LIN {X 0,Y 148.489,Z 220.439,A -85,B 0,C 180,E1 -25225.922,E2 -25225.922} C_VEL
LIN {X 0,Y 152.056,Z 225.38,A -85,B 0,C 180,E1 -25229.033,E2 -25229.033} C_VEL
LIN {X 0,Y 155.13,Z 229.793,A -85,B 0,C 180,E1 -25231.399,E2 -25231.399} C_VEL
LIN {X 0,Y 159.463,Z 236.417,A -85,B 0,C 180,E1 -25234.38,E2 -25234.38} C_VEL
LIN {X 0,Y 163.977,Z 245.373,A -85,B 0,C 180,E1 -25237.257,E2 -25237.257} C_VEL
LIN {X 0,Y 168.416,Z 255.821,A -85,B 0,C 180,E1 -25239.882,E2 -25239.882} C_VEL
LIN {X 0,Y 170.789,Z 262.4,A -85,B 0,C 180,E1 -25241.237,E2 -25241.237} C_VEL
LIN {X 0,Y 168.029,Z 299.799,A -85,B 0,C 180,E1 -25242.631,E2 -25242.631} C_VEL
LIN {X 0,Y 166.027,Z 312.888,A -85,B 0,C 180,E1 -25243.453,E2 -25243.453} C_VEL
LIN {X 0,Y 163.042,Z 325.855,A -85,B 0,C 180,E1 -25244.664,E2 -25244.664} C_VEL
LIN {X 0,Y 159.734,Z 336.912,A -85,B 0,C 180,E1 -25246.134,E2 -25246.134} C_VEL
LIN {X 0,Y 155.587,Z 348.447,A -85,B 0,C 180,E1 -25248.22,E2 -25248.22} C_VEL
LIN {X 0,Y 151.08,Z 358.834,A -85,B 0,C 180,E1 -25250.668,E2 -25250.668} C_VEL
LIN {X 0,Y 146.904,Z 367.324,A -85,B 0,C 180,E1 -25253.272,E2 -25253.272} C_VEL
LIN {X 0,Y 142.719,Z 375.157,A -85,B 0,C 180,E1 -25256.358,E2 -25256.358} C_VEL
LIN {X 0,Y 138.407,Z 382.806,A -85,B 0,C 180,E1 -25260.324,E2 -25260.324} C_VEL
LIN {X 0,Y 135.143,Z 388.047,A -85,B 0,C 180,E1 -25263.765,E2 -25263.765} C_VEL
LIN {X 0,Y 131.795,Z 393.123,A -85,B 0,C 180,E1 -25268.081,E2 -25268.081} C_VEL
LIN {X 0,Y 129.336,Z 397.065,A -85,B 0,C 180,E1 -25272.61,E2 -25272.61} C_VEL
LIN {X 0,Y 127.624,Z 399.977,A -85,B 0,C 180,E1 -25277.274,E2 -25277.274} C_VEL
LIN {X 0,Y 126.711,Z 401.714,A -85,B 0,C 180,E1 -25281.57,E2 -25281.57} C_VEL
LIN {X 0,Y 126.307,Z 402.951,A -85,B 0,C 180,E1 -25286.809,E2 -25286.809} C_VEL
LIN {X 0,Y 126.321,Z 403.159,A -85,B 0,C 180,E1 -25289.999,E2 -25289.999} C_VEL
LIN {X 0,Y 126.384,Z 402.517,A -85,B 0,C 180,E1 -25295.368,E2 -25295.368} C_VEL
LIN {X 0,Y 126.011,Z 401.88,A -85,B 0,C 180,E1 -25298.026,E2 -25298.026} C_VEL
LIN {X 0,Y 124.021,Z 400.249,A -85,B 0,C 180,E1 -25302.416,E2 -25302.416} C_VEL
LIN {X 0,Y 122.691,Z 398.422,A -85,B 0,C 180,E1 -25305.973,E2 -25305.973} C_VEL
LIN {X 0,Y 122.726,Z 396.742,A -85,B 0,C 180,E1 -25308.632,E2 -25308.632} C_VEL
LIN {X 0,Y 123.046,Z 396.081,A -85,B 0,C 180,E1 -25309.494,E2 -25309.494} C_VEL
LIN {X 0,Y 126.316,Z 391.361,A -85,B 0,C 180,E1 -25314.661,E2 -25314.661} C_VEL
LIN {X 0,Y 130.041,Z 385.839,A -85,B 0,C 180,E1 -25319.102,E2 -25319.102} C_VEL
LIN {X 0,Y 134.152,Z 379.389,A -85,B 0,C 180,E1 -25323.048,E2 -25323.048} C_VEL
LIN {X 0,Y 138.51,Z 371.906,A -85,B 0,C 180,E1 -25326.595,E2 -25326.595} C_VEL
LIN {X 0,Y 143.179,Z 363.415,A -85,B 0,C 180,E1 -25329.648,E2 -25329.648} C_VEL
LIN {X 0,Y 148.185,Z 352.923,A -85,B 0,C 180,E1 -25332.516,E2 -25332.516} C_VEL
LIN {X 0,Y 152.513,Z 342.536,A -85,B 0,C 180,E1 -25334.644,E2 -25334.644} C_VEL
LIN {X 0,Y 156.431,Z 331.134,A -85,B 0,C 180,E1 -25336.42,E2 -25336.42} C_VEL
LIN {X 0,Y 159.575,Z 319.369,A -85,B 0,C 180,E1 -25337.767,E2 -25337.767} C_VEL
LIN {X 0,Y 162.297,Z 305.659,A -85,B 0,C 180,E1 -25338.812,E2 -25338.812} C_VEL
LIN {X 0,Y 163.803,Z 292.635,A -85,B 0,C 180,E1 -25339.441,E2 -25339.441} C_VEL
LIN {X 0,Y 165.84,Z 264.469,A -85,B 0,C 180,E1 -25340.466,E2 -25340.466} C_VEL
LIN {X 0,Y 162.183,Z 254.665,A -85,B 0,C 180,E1 -25342.749,E2 -25342.749} C_VEL
LIN {X 0,Y 157.734,Z 244.687,A -85,B 0,C 180,E1 -25345.703,E2 -25345.703} C_VEL
LIN {X 0,Y 155.11,Z 239.926,A -85,B 0,C 180,E1 -25347.545,E2 -25347.545} C_VEL
LIN {X 0,Y 150.936,Z 233.432,A -85,B 0,C 180,E1 -25350.731,E2 -25350.731} C_VEL
LIN {X 0,Y 148.33,Z 229.665,A -85,B 0,C 180,E1 -25352.963,E2 -25352.963} C_VEL
LIN {X 0,Y 145.763,Z 225.988,A -85,B 0,C 180,E1 -25355.427,E2 -25355.427} C_VEL
LIN {X 0,Y 142.909,Z 222.259,A -85,B 0,C 180,E1 -25358.546,E2 -25358.546} C_VEL
LIN {X 0,Y 142.242,Z 221.258,A -85,B 0,C 180,E1 -25359.376,E2 -25359.376} C_VEL
LIN {X 0,Y 139.642,Z 218.363,A -85,B 0,C 180,E1 -25362.898,E2 -25362.898} C_VEL
LIN {X 0,Y 138.606,Z 216.213,A -85,B 0,C 180,E1 -25364.75,E2 -25364.75} C_VEL
LIN {X 0,Y 136.107,Z 214.124,A -85,B 0,C 180,E1 -25369.815,E2 -25369.815} C_VEL
LIN {X 0,Y 134.66,Z 211.097,A -85,B 0,C 180,E1 -25375.885,E2 -25375.885} C_VEL
LIN {X 0,Y 134.387,Z 210.372,A -85,B 0,C 180,E1 -25380,E2 -25380} C_VEL
LIN {X 0,Y 134.78,Z 211.442,A -85,B 0,C 180,E1 -25385.142,E2 -25385.142} C_VEL
LIN {X 0,Y 137.586,Z 215.64,A -85,B 0,C 180,E1 -25393.665,E2 -25393.665} C_VEL
LIN {X 0,Y 138.782,Z 216.531,A -85,B 0,C 180,E1 -25395.747,E2 -25395.747} C_VEL
LIN {X 0,Y 140.767,Z 219.894,A -85,B 0,C 180,E1 -25398.937,E2 -25398.937} C_VEL
LIN {X 0,Y 142.714,Z 221.837,A -85,B 0,C 180,E1 -25401.372,E2 -25401.372} C_VEL
LIN {X 0,Y 145.287,Z 225.513,A -85,B 0,C 180,E1 -25404.279,E2 -25404.279} C_VEL
LIN {X 0,Y 146.423,Z 226.871,A -85,B 0,C 180,E1 -25405.403,E2 -25405.403} C_VEL
LIN {X 0,Y 149.767,Z 231.675,A -85,B 0,C 180,E1 -25408.464,E2 -25408.464} C_VEL
LIN {X 0,Y 152.784,Z 236.265,A -85,B 0,C 180,E1 -25410.908,E2 -25410.908} C_VEL
LIN {X 0,Y 156.375,Z 241.912,A -85,B 0,C 180,E1 -25413.51,E2 -25413.51} C_VEL
LIN {X 0,Y 161.078,Z 250.32,A -85,B 0,C 180,E1 -25416.588,E2 -25416.588} C_VEL
LIN {X 0,Y 164.621,Z 258.823,A -85,B 0,C 180,E1 -25418.808,E2 -25418.808} C_VEL
LIN {X 0,Y 165.991,Z 262.553,A -85,B 0,C 180,E1 -25419.643,E2 -25419.643} C_VEL
LIN {X 0,Y 163.242,Z 297.955,A -85,B 0,C 180,E1 -25420.978,E2 -25420.978} C_VEL
LIN {X 0,Y 161.003,Z 311.512,A -85,B 0,C 180,E1 -25421.82,E2 -25421.82} C_VEL
LIN {X 0,Y 158.165,Z 324.036,A -85,B 0,C 180,E1 -25423.084,E2 -25423.084} C_VEL
LIN {X 0,Y 154.484,Z 335.831,A -85,B 0,C 180,E1 -25424.7,E2 -25424.7} C_VEL
LIN {X 0,Y 150.193,Z 347.172,A -85,B 0,C 180,E1 -25426.818,E2 -25426.818} C_VEL
LIN {X 0,Y 145.558,Z 357.394,A -85,B 0,C 180,E1 -25429.324,E2 -25429.324} C_VEL
LIN {X 0,Y 140.81,Z 366.572,A -85,B 0,C 180,E1 -25432.311,E2 -25432.311} C_VEL
LIN {X 0,Y 135.827,Z 375.493,A -85,B 0,C 180,E1 -25436.207,E2 -25436.207} C_VEL
LIN {X 0,Y 131.307,Z 382.676,A -85,B 0,C 180,E1 -25440.326,E2 -25440.326} C_VEL
LIN {X 0,Y 127.933,Z 387.52,A -85,B 0,C 180,E1 -25443.931,E2 -25443.931} C_VEL
LIN {X 0,Y 124.651,Z 392.227,A -85,B 0,C 180,E1 -25448.503,E2 -25448.503} C_VEL
LIN {X 0,Y 122.223,Z 395.828,A -85,B 0,C 180,E1 -25453.293,E2 -25453.293} C_VEL
LIN {X 0,Y 120.997,Z 397.687,A -85,B 0,C 180,E1 -25456.567,E2 -25456.567} C_VEL
LIN {X 0,Y 120.126,Z 399.083,A -85,B 0,C 180,E1 -25459.893,E2 -25459.893} C_VEL
LIN {X 0,Y 119.293,Z 400.686,A -85,B 0,C 180,E1 -25466.624,E2 -25466.624} C_VEL
LIN {X 0,Y 119.281,Z 400.912,A -85,B 0,C 180,E1 -25470.001,E2 -25470.001} C_VEL
LIN {X 0,Y 119.293,Z 400.715,A -85,B 0,C 180,E1 -25473.379,E2 -25473.379} C_VEL
LIN {X 0,Y 120.127,Z 399.15,A -85,B 0,C 180,E1 -25480.11,E2 -25480.11} C_VEL
LIN {X 0,Y 120.997,Z 397.783,A -85,B 0,C 180,E1 -25483.436,E2 -25483.436} C_VEL
LIN {X 0,Y 122.934,Z 394.897,A -85,B 0,C 180,E1 -25488.327,E2 -25488.327} C_VEL
LIN {X 0,Y 125.547,Z 390.986,A -85,B 0,C 180,E1 -25493.071,E2 -25493.071} C_VEL
LIN {X 0,Y 129.152,Z 385.94,A -85,B 0,C 180,E1 -25497.552,E2 -25497.552} C_VEL
LIN {X 0,Y 133.341,Z 379.586,A -85,B 0,C 180,E1 -25501.808,E2 -25501.808} C_VEL
LIN {X 0,Y 138.101,Z 371.645,A -85,B 0,C 180,E1 -25505.819,E2 -25505.819} C_VEL
LIN {X 0,Y 142.511,Z 363.544,A -85,B 0,C 180,E1 -25508.96,E2 -25508.96} C_VEL
LIN {X 0,Y 147.519,Z 353.661,A -85,B 0,C 180,E1 -25511.835,E2 -25511.835} C_VEL
LIN {X 0,Y 152.249,Z 342.531,A -85,B 0,C 180,E1 -25514.282,E2 -25514.282} C_VEL
LIN {X 0,Y 156.034,Z 331.622,A -85,B 0,C 180,E1 -25516.109,E2 -25516.109} C_VEL
LIN {X 0,Y 159.484,Z 319.56,A -85,B 0,C 180,E1 -25517.572,E2 -25517.572} C_VEL
LIN {X 0,Y 162.175,Z 306.48,A -85,B 0,C 180,E1 -25518.694,E2 -25518.694} C_VEL
LIN {X 0,Y 163.866,Z 293.691,A -85,B 0,C 180,E1 -25519.374,E2 -25519.374} C_VEL
LIN {X 0,Y 166.138,Z 262.629,A -85,B 0,C 180,E1 -25520.526,E2 -25520.526} C_VEL
LIN {X 0,Y 162.62,Z 253.552,A -85,B 0,C 180,E1 -25522.703,E2 -25522.703} C_VEL
LIN {X 0,Y 159.851,Z 247.737,A -85,B 0,C 180,E1 -25524.466,E2 -25524.466} C_VEL
LIN {X 0,Y 154.056,Z 237.994,A -85,B 0,C 180,E1 -25528.452,E2 -25528.452} C_VEL
LIN {X 0,Y 149.123,Z 230.481,A -85,B 0,C 180,E1 -25532.454,E2 -25532.454} C_VEL
LIN {X 0,Y 145.784,Z 225.926,A -85,B 0,C 180,E1 -25535.62,E2 -25535.62} C_VEL
LIN {X 0,Y 143.1,Z 222.493,A -85,B 0,C 180,E1 -25538.575,E2 -25538.575} C_VEL
LIN {X 0,Y 142.318,Z 221.292,A -85,B 0,C 180,E1 -25539.564,E2 -25539.564} C_VEL
LIN {X 0,Y 139.639,Z 218.207,A -85,B 0,C 180,E1 -25543.296,E2 -25543.296} C_VEL
LIN {X 0,Y 138.742,Z 216.293,A -85,B 0,C 180,E1 -25544.953,E2 -25544.953} C_VEL
LIN {X 0,Y 135.941,Z 213.85,A -85,B 0,C 180,E1 -25551.077,E2 -25551.077} C_VEL
LIN {X 0,Y 134.761,Z 210.99,A -85,B 0,C 180,E1 -25557.758,E2 -25557.758} C_VEL
LIN {X 0,Y 134.713,Z 210.681,A -85,B 0,C 180,E1 -25560.747,E2 -25560.747} C_VEL
LIN {X 0,Y 134.979,Z 211.831,A -85,B 0,C 180,E1 -25564.479,E2 -25564.479} C_VEL
LIN {X 0,Y 137.967,Z 215.899,A -85,B 0,C 180,E1 -25573.627,E2 -25573.627} C_VEL
LIN {X 0,Y 138.803,Z 216.447,A -85,B 0,C 180,E1 -25575.087,E2 -25575.087} C_VEL
LIN {X 0,Y 140.718,Z 219.788,A -85,B 0,C 180,E1 -25578.283,E2 -25578.283} C_VEL
LIN {X 0,Y 142.808,Z 221.926,A -85,B 0,C 180,E1 -25580.962,E2 -25580.962} C_VEL
LIN {X 0,Y 145.247,Z 225.428,A -85,B 0,C 180,E1 -25583.764,E2 -25583.764} C_VEL
LIN {X 0,Y 146.569,Z 227.031,A -85,B 0,C 180,E1 -25585.091,E2 -25585.091} C_VEL
LIN {X 0,Y 149.847,Z 231.734,A -85,B 0,C 180,E1 -25588.114,E2 -25588.114} C_VEL
LIN {X 0,Y 153.25,Z 236.86,A -85,B 0,C 180,E1 -25590.868,E2 -25590.868} C_VEL
LIN {X 0,Y 157.046,Z 243.057,A -85,B 0,C 180,E1 -25593.612,E2 -25593.612} C_VEL
LIN {X 0,Y 161.42,Z 252.589,A -85,B 0,C 180,E1 -25596.579,E2 -25596.579} C_VEL
LIN {X 0,Y 165.179,Z 262.134,A -85,B 0,C 180,E1 -25598.95,E2 -25598.95} C_VEL
LIN {X 0,Y 166.024,Z 264.644,A -85,B 0,C 180,E1 -25599.476,E2 -25599.476} C_VEL
LIN {X 0,Y 163.281,Z 299.957,A -85,B 0,C 180,E1 -25600.81,E2 -25600.81} C_VEL
LIN {X 0,Y 161.16,Z 313.156,A -85,B 0,C 180,E1 -25601.644,E2 -25601.644} C_VEL
LIN {X 0,Y 158.144,Z 325.797,A -85,B 0,C 180,E1 -25602.839,E2 -25602.839} C_VEL
LIN {X 0,Y 154.699,Z 336.852,A -85,B 0,C 180,E1 -25604.314,E2 -25604.314} C_VEL
LIN {X 0,Y 150.368,Z 348.386,A -85,B 0,C 180,E1 -25606.418,E2 -25606.418} C_VEL
LIN {X 0,Y 145.665,Z 358.772,A -85,B 0,C 180,E1 -25608.9,E2 -25608.9} C_VEL
LIN {X 0,Y 141.276,Z 367.262,A -85,B 0,C 180,E1 -25611.55,E2 -25611.55} C_VEL
LIN {X 0,Y 136.015,Z 376.462,A -85,B 0,C 180,E1 -25615.362,E2 -25615.362} C_VEL
LIN {X 0,Y 131.525,Z 383.859,A -85,B 0,C 180,E1 -25619.493,E2 -25619.493} C_VEL
LIN {X 0,Y 127.531,Z 389.797,A -85,B 0,C 180,E1 -25623.84,E2 -25623.84} C_VEL
LIN {X 0,Y 124.214,Z 394.486,A -85,B 0,C 180,E1 -25628.421,E2 -25628.421} C_VEL
LIN {X 0,Y 121.847,Z 398.067,A -85,B 0,C 180,E1 -25633.237,E2 -25633.237} C_VEL
LIN {X 0,Y 120.689,Z 399.913,A -85,B 0,C 180,E1 -25636.529,E2 -25636.529} C_VEL
LIN {X 0,Y 119.43,Z 402.284,A -85,B 0,C 180,E1 -25643.24,E2 -25643.24} C_VEL
LIN {X 0,Y 119.225,Z 402.886,A -85,B 0,C 180,E1 -25646.619,E2 -25646.619} C_VEL
LIN {X 0,Y 119.234,Z 403.094,A -85,B 0,C 180,E1 -25649.999,E2 -25649.999} C_VEL
LIN {X 0,Y 119.303,Z 402.488,A -85,B 0,C 180,E1 -25655.484,E2 -25655.484} C_VEL
LIN {X 0,Y 119.887,Z 401.259,A -85,B 0,C 180,E1 -25660.127,E2 -25660.127} C_VEL
LIN {X 0,Y 120.704,Z 399.859,A -85,B 0,C 180,E1 -25663.466,E2 -25663.466} C_VEL
LIN {X 0,Y 123.046,Z 396.081,A -85,B 0,C 180,E1 -25669.494,E2 -25669.494} C_VEL
LIN {X 0,Y 123.774,Z 394.072,A -85,B 0,C 180,E1 -25672.05,E2 -25672.05} C_VEL
LIN {X 0,Y 123.81,Z 390.329,A -85,B 0,C 180,E1 -25676.3,E2 -25676.3} C_VEL
LIN {X 0,Y 124.391,Z 385.968,A -85,B 0,C 180,E1 -25680.398,E2 -25680.398} C_VEL
LIN {X 0,Y 125.914,Z 382.924,A -85,B 0,C 180,E1 -25682.618,E2 -25682.618} C_VEL
LIN {X 0,Y 131.063,Z 374.812,A -85,B 0,C 180,E1 -25687.101,E2 -25687.101} C_VEL
LIN {X 0,Y 135.761,Z 366.932,A -85,B 0,C 180,E1 -25690.32,E2 -25690.32} C_VEL
LIN {X 0,Y 140.867,Z 357.317,A -85,B 0,C 180,E1 -25693.311,E2 -25693.311} C_VEL
LIN {X 0,Y 145.774,Z 346.644,A -85,B 0,C 180,E1 -25695.816,E2 -25695.816} C_VEL
LIN {X 0,Y 149.829,Z 336.315,A -85,B 0,C 180,E1 -25697.625,E2 -25697.625} C_VEL
LIN {X 0,Y 153.705,Z 323.946,A -85,B 0,C 180,E1 -25699.224,E2 -25699.224} C_VEL
LIN {X 0,Y 156.725,Z 311.132,A -85,B 0,C 180,E1 -25700.38,E2 -25700.38} C_VEL
LIN {X 0,Y 158.79,Z 297.868,A -85,B 0,C 180,E1 -25701.159,E2 -25701.159} C_VEL
LIN {X 0,Y 161.234,Z 266.782,A -85,B 0,C 180,E1 -25702.322,E2 -25702.322} C_VEL
LIN {X 0,Y 157.654,Z 257.066,A -85,B 0,C 180,E1 -25704.778,E2 -25704.778} C_VEL
LIN {X 0,Y 153.773,Z 248.275,A -85,B 0,C 180,E1 -25707.616,E2 -25707.616} C_VEL
LIN {X 0,Y 150.126,Z 242.029,A -85,B 0,C 180,E1 -25710.46,E2 -25710.46} C_VEL
LIN {X 0,Y 146.642,Z 236.472,A -85,B 0,C 180,E1 -25713.541,E2 -25713.541} C_VEL
LIN {X 0,Y 143.63,Z 232.219,A -85,B 0,C 180,E1 -25716.574,E2 -25716.574} C_VEL
LIN {X 0,Y 140.558,Z 227.87,A -85,B 0,C 180,E1 -25720.275,E2 -25720.275} C_VEL
LIN {X 0,Y 137.868,Z 224.441,A -85,B 0,C 180,E1 -25724.287,E2 -25724.287} C_VEL
LIN {X 0,Y 137.228,Z 223.045,A -85,B 0,C 180,E1 -25725.542,E2 -25725.542} C_VEL
LIN {X 0,Y 134.693,Z 220.54,A -85,B 0,C 180,E1 -25731.373,E2 -25731.373} C_VEL
LIN {X 0,Y 133.719,Z 218.034,A -85,B 0,C 180,E1 -25736.422,E2 -25736.422} C_VEL
LIN {X 0,Y 133.52,Z 217.429,A -85,B 0,C 180,E1 -25740,E2 -25740} C_VEL
LIN {X 0,Y 133.863,Z 218.47,A -85,B 0,C 180,E1 -25744.894,E2 -25744.894} C_VEL
LIN {X 0,Y 136.363,Z 222.503,A -85,B 0,C 180,E1 -25753.031,E2 -25753.031} C_VEL
LIN {X 0,Y 137.429,Z 223.408,A -85,B 0,C 180,E1 -25755.023,E2 -25755.023} C_VEL
LIN {X 0,Y 139.535,Z 226.869,A -85,B 0,C 180,E1 -25758.539,E2 -25758.539} C_VEL
LIN {X 0,Y 141.056,Z 228.526,A -85,B 0,C 180,E1 -25760.547,E2 -25760.547} C_VEL
LIN {X 0,Y 143.805,Z 232.367,A -85,B 0,C 180,E1 -25763.778,E2 -25763.778} C_VEL
LIN {X 0,Y 147.492,Z 237.884,A -85,B 0,C 180,E1 -25767.434,E2 -25767.434} C_VEL
LIN {X 0,Y 150.332,Z 242.336,A -85,B 0,C 180,E1 -25769.88,E2 -25769.88} C_VEL
LIN {X 0,Y 155.024,Z 250.278,A -85,B 0,C 180,E1 -25773.443,E2 -25773.443} C_VEL
LIN {X 0,Y 158.233,Z 256.652,A -85,B 0,C 180,E1 -25775.659,E2 -25775.659} C_VEL
LIN {X 0,Y 161.38,Z 264.879,A -85,B 0,C 180,E1 -25777.784,E2 -25777.784} C_VEL
LIN {X 0,Y 158.734,Z 297.656,A -85,B 0,C 180,E1 -25779.026,E2 -25779.026} C_VEL
LIN {X 0,Y 156.442,Z 311.248,A -85,B 0,C 180,E1 -25779.862,E2 -25779.862} C_VEL
LIN {X 0,Y 153.411,Z 324.107,A -85,B 0,C 180,E1 -25781.15,E2 -25781.15} C_VEL
LIN {X 0,Y 149.581,Z 335.901,A -85,B 0,C 180,E1 -25782.769,E2 -25782.769} C_VEL
LIN {X 0,Y 145.106,Z 347.241,A -85,B 0,C 180,E1 -25784.903,E2 -25784.903} C_VEL
LIN {X 0,Y 140.253,Z 357.463,A -85,B 0,C 180,E1 -25787.434,E2 -25787.434} C_VEL
LIN {X 0,Y 135.256,Z 366.64,A -85,B 0,C 180,E1 -25790.47,E2 -25790.47} C_VEL
LIN {X 0,Y 130.16,Z 375.252,A -85,B 0,C 180,E1 -25794.304,E2 -25794.304} C_VEL
LIN {X 0,Y 125.175,Z 382.743,A -85,B 0,C 180,E1 -25798.714,E2 -25798.714} C_VEL
LIN {X 0,Y 121.578,Z 387.587,A -85,B 0,C 180,E1 -25802.457,E2 -25802.457} C_VEL
LIN {X 0,Y 118.039,Z 392.294,A -85,B 0,C 180,E1 -25807.234,E2 -25807.234} C_VEL
LIN {X 0,Y 115.428,Z 395.894,A -85,B 0,C 180,E1 -25812.278,E2 -25812.278} C_VEL
LIN {X 0,Y 114.081,Z 397.753,A -85,B 0,C 180,E1 -25815.736,E2 -25815.736} C_VEL
LIN {X 0,Y 113.129,Z 399.148,A -85,B 0,C 180,E1 -25819.261,E2 -25819.261} C_VEL
LIN {X 0,Y 112.213,Z 400.751,A -85,B 0,C 180,E1 -25826.411,E2 -25826.411} C_VEL
LIN {X 0,Y 112.2,Z 400.977,A -85,B 0,C 180,E1 -25830.002,E2 -25830.002} C_VEL
LIN {X 0,Y 112.213,Z 400.78,A -85,B 0,C 180,E1 -25833.592,E2 -25833.592} C_VEL
LIN {X 0,Y 113.129,Z 399.215,A -85,B 0,C 180,E1 -25840.742,E2 -25840.742} C_VEL
LIN {X 0,Y 114.081,Z 397.848,A -85,B 0,C 180,E1 -25844.267,E2 -25844.267} C_VEL
LIN {X 0,Y 116.19,Z 394.962,A -85,B 0,C 180,E1 -25849.433,E2 -25849.433} C_VEL
LIN {X 0,Y 119.034,Z 391.05,A -85,B 0,C 180,E1 -25854.413,E2 -25854.413} C_VEL
LIN {X 0,Y 122.896,Z 386.003,A -85,B 0,C 180,E1 -25859.084,E2 -25859.084} C_VEL
LIN {X 0,Y 127.368,Z 379.649,A -85,B 0,C 180,E1 -25863.49,E2 -25863.49} C_VEL
LIN {X 0,Y 132.384,Z 371.704,A -85,B 0,C 180,E1 -25867.627,E2 -25867.627} C_VEL
LIN {X 0,Y 137.066,Z 363.606,A -85,B 0,C 180,E1 -25870.826,E2 -25870.826} C_VEL
LIN {X 0,Y 142.291,Z 353.723,A -85,B 0,C 180,E1 -25873.748,E2 -25873.748} C_VEL
LIN {X 0,Y 147.252,Z 342.591,A -85,B 0,C 180,E1 -25876.21,E2 -25876.21} C_VEL
LIN {X 0,Y 151.206,Z 331.682,A -85,B 0,C 180,E1 -25878.046,E2 -25878.046} C_VEL
LIN {X 0,Y 154.775,Z 319.618,A -85,B 0,C 180,E1 -25879.516,E2 -25879.516} C_VEL
LIN {X 0,Y 157.562,Z 306.663,A -85,B 0,C 180,E1 -25880.623,E2 -25880.623} C_VEL
LIN {X 0,Y 159.349,Z 293.381,A -85,B 0,C 180,E1 -25881.335,E2 -25881.335} C_VEL
LIN {X 0,Y 161.54,Z 264.943,A -85,B 0,C 180,E1 -25882.388,E2 -25882.388} C_VEL
LIN {X 0,Y 157.819,Z 255.359,A -85,B 0,C 180,E1 -25884.918,E2 -25884.918} C_VEL
LIN {X 0,Y 153.237,Z 246.935,A -85,B 0,C 180,E1 -25888.168,E2 -25888.168} C_VEL
LIN {X 0,Y 148.476,Z 239.258,A -85,B 0,C 180,E1 -25892.036,E2 -25892.036} C_VEL
LIN {X 0,Y 146.101,Z 235.699,A -85,B 0,C 180,E1 -25894.24,E2 -25894.24} C_VEL
LIN {X 0,Y 143.821,Z 232.339,A -85,B 0,C 180,E1 -25896.607,E2 -25896.607} C_VEL
LIN {X 0,Y 141.03,Z 228.357,A -85,B 0,C 180,E1 -25899.964,E2 -25899.964} C_VEL
LIN {X 0,Y 138.048,Z 224.594,A -85,B 0,C 180,E1 -25904.403,E2 -25904.403} C_VEL
LIN {X 0,Y 137.378,Z 223.109,A -85,B 0,C 180,E1 -25905.747,E2 -25905.747} C_VEL
LIN {X 0,Y 134.751,Z 220.492,A -85,B 0,C 180,E1 -25912.131,E2 -25912.131} C_VEL
LIN {X 0,Y 133.891,Z 218.08,A -85,B 0,C 180,E1 -25917.744,E2 -25917.744} C_VEL
LIN {X 0,Y 133.845,Z 217.746,A -85,B 0,C 180,E1 -25920.752,E2 -25920.752} C_VEL
LIN {X 0,Y 134.151,Z 219.184,A -85,B 0,C 180,E1 -25924.883,E2 -25924.883} C_VEL
LIN {X 0,Y 136.929,Z 222.866,A -85,B 0,C 180,E1 -25933.354,E2 -25933.354} C_VEL
LIN {X 0,Y 137.544,Z 223.498,A -85,B 0,C 180,E1 -25934.518,E2 -25934.518} C_VEL
LIN {X 0,Y 139.554,Z 226.828,A -85,B 0,C 180,E1 -25937.966,E2 -25937.966} C_VEL
LIN {X 0,Y 141.146,Z 228.577,A -85,B 0,C 180,E1 -25940.113,E2 -25940.113} C_VEL
LIN {X 0,Y 143.734,Z 232.244,A -85,B 0,C 180,E1 -25943.217,E2 -25943.217} C_VEL
LIN {X 0,Y 147.59,Z 237.946,A -85,B 0,C 180,E1 -25947.087,E2 -25947.087} C_VEL
LIN {X 0,Y 151.393,Z 243.842,A -85,B 0,C 180,E1 -25950.321,E2 -25950.321} C_VEL
LIN {X 0,Y 154.182,Z 248.936,A -85,B 0,C 180,E1 -25952.481,E2 -25952.481} C_VEL
LIN {X 0,Y 157.857,Z 257.311,A -85,B 0,C 180,E1 -25955.169,E2 -25955.169} C_VEL
LIN {X 0,Y 161.263,Z 266.348,A -85,B 0,C 180,E1 -25957.501,E2 -25957.501} C_VEL
LIN {X 0,Y 161.479,Z 267.017,A -85,B 0,C 180,E1 -25957.648,E2 -25957.648} C_VEL
LIN {X 0,Y 158.755,Z 299.84,A -85,B 0,C 180,E1 -25958.873,E2 -25958.873} C_VEL
LIN {X 0,Y 156.464,Z 313.428,A -85,B 0,C 180,E1 -25959.726,E2 -25959.726} C_VEL
LIN {X 0,Y 153.413,Z 325.738,A -85,B 0,C 180,E1 -25960.897,E2 -25960.897} C_VEL
LIN {X 0,Y 149.228,Z 338.374,A -85,B 0,C 180,E1 -25962.619,E2 -25962.619} C_VEL
LIN {X 0,Y 144.763,Z 349.618,A -85,B 0,C 180,E1 -25964.763,E2 -25964.763} C_VEL
LIN {X 0,Y 139.86,Z 359.74,A -85,B 0,C 180,E1 -25967.282,E2 -25967.282} C_VEL
LIN {X 0,Y 134.81,Z 368.862,A -85,B 0,C 180,E1 -25970.31,E2 -25970.31} C_VEL
LIN {X 0,Y 129.465,Z 377.601,A -85,B 0,C 180,E1 -25974.189,E2 -25974.189} C_VEL
LIN {X 0,Y 124.666,Z 384.906,A -85,B 0,C 180,E1 -25978.569,E2 -25978.569} C_VEL
LIN {X 0,Y 119.893,Z 391.415,A -85,B 0,C 180,E1 -25983.918,E2 -25983.918} C_VEL
LIN {X 0,Y 116.622,Z 395.721,A -85,B 0,C 180,E1 -25988.802,E2 -25988.802} C_VEL
LIN {X 0,Y 115.053,Z 398.003,A -85,B 0,C 180,E1 -25992.215,E2 -25992.215} C_VEL
LIN {X 0,Y 113.772,Z 399.848,A -85,B 0,C 180,E1 -25995.693,E2 -25995.693} C_VEL
LIN {X 0,Y 112.36,Z 402.22,A -85,B 0,C 180,E1 -26002.812,E2 -26002.812} C_VEL
LIN {X 0,Y 112.135,Z 402.822,A -85,B 0,C 180,E1 -26006.405,E2 -26006.405} C_VEL
LIN {X 0,Y 112.139,Z 403.03,A -85,B 0,C 180,E1 -26009.998,E2 -26009.998} C_VEL
LIN {X 0,Y 112.135,Z 402.805,A -85,B 0,C 180,E1 -26013.592,E2 -26013.592} C_VEL
LIN {X 0,Y 112.359,Z 402.192,A -85,B 0,C 180,E1 -26017.185,E2 -26017.185} C_VEL
LIN {X 0,Y 112.895,Z 401.193,A -85,B 0,C 180,E1 -26020.762,E2 -26020.762} C_VEL
LIN {X 0,Y 113.784,Z 399.793,A -85,B 0,C 180,E1 -26024.302,E2 -26024.302} C_VEL
LIN {X 0,Y 116.164,Z 396.283,A -85,B 0,C 180,E1 -26030.296,E2 -26030.296} C_VEL
LIN {X 0,Y 119.885,Z 391.294,A -85,B 0,C 180,E1 -26036.08,E2 -26036.08} C_VEL
LIN {X 0,Y 123.881,Z 385.773,A -85,B 0,C 180,E1 -26040.7,E2 -26040.7} C_VEL
LIN {X 0,Y 125.914,Z 382.924,A -85,B 0,C 180,E1 -26042.618,E2 -26042.618} C_VEL
LIN {X 0,Y 127.508,Z 379.706,A -85,B 0,C 180,E1 -26044.738,E2 -26044.738} C_VEL
LIN {X 0,Y 128.744,Z 374.105,A -85,B 0,C 180,E1 -26048.355,E2 -26048.355} C_VEL
LIN {X 0,Y 130.262,Z 368.002,A -85,B 0,C 180,E1 -26051.719,E2 -26051.719} C_VEL
LIN {X 0,Y 132.2,Z 363.87,A -85,B 0,C 180,E1 -26053.37,E2 -26053.37} C_VEL
LIN {X 0,Y 137.478,Z 353.96,A -85,B 0,C 180,E1 -26056.224,E2 -26056.224} C_VEL
LIN {X 0,Y 142.164,Z 343.824,A -85,B 0,C 180,E1 -26058.39,E2 -26058.39} C_VEL
LIN {X 0,Y 146.387,Z 332.763,A -85,B 0,C 180,E1 -26060.185,E2 -26060.185} C_VEL
LIN {X 0,Y 150.098,Z 320.479,A -85,B 0,C 180,E1 -26061.651,E2 -26061.651} C_VEL
LIN {X 0,Y 153.106,Z 306.849,A -85,B 0,C 180,E1 -26062.715,E2 -26062.715} C_VEL
LIN {X 0,Y 154.809,Z 293.931,A -85,B 0,C 180,E1 -26063.375,E2 -26063.375} C_VEL
LIN {X 0,Y 156.789,Z 269.085,A -85,B 0,C 180,E1 -26064.294,E2 -26064.294} C_VEL
LIN {X 0,Y 153.223,Z 259.353,A -85,B 0,C 180,E1 -26066.997,E2 -26066.997} C_VEL
LIN {X 0,Y 150.007,Z 252.084,A -85,B 0,C 180,E1 -26069.598,E2 -26069.598} C_VEL
LIN {X 0,Y 145.981,Z 245.196,A -85,B 0,C 180,E1 -26073.122,E2 -26073.122} C_VEL
LIN {X 0,Y 142.959,Z 240.534,A -85,B 0,C 180,E1 -26076.169,E2 -26076.169} C_VEL
LIN {X 0,Y 141.47,Z 238.323,A -85,B 0,C 180,E1 -26077.857,E2 -26077.857} C_VEL
LIN {X 0,Y 138.858,Z 234.383,A -85,B 0,C 180,E1 -26081.272,E2 -26081.272} C_VEL
LIN {X 0,Y 136.307,Z 230.794,A -85,B 0,C 180,E1 -26085.442,E2 -26085.442} C_VEL
LIN {X 0,Y 135.781,Z 229.827,A -85,B 0,C 180,E1 -26086.531,E2 -26086.531} C_VEL
LIN {X 0,Y 133.336,Z 226.789,A -85,B 0,C 180,E1 -26093.189,E2 -26093.189} C_VEL
LIN {X 0,Y 132.79,Z 224.977,A -85,B 0,C 180,E1 -26096.966,E2 -26096.966} C_VEL
LIN {X 0,Y 132.654,Z 224.485,A -85,B 0,C 180,E1 -26100,E2 -26100} C_VEL
LIN {X 0,Y 132.888,Z 225.327,A -85,B 0,C 180,E1 -26104.17,E2 -26104.17} C_VEL
LIN {X 0,Y 135.331,Z 229.497,A -85,B 0,C 180,E1 -26112.751,E2 -26112.751} C_VEL
LIN {X 0,Y 136.149,Z 230.361,A -85,B 0,C 180,E1 -26114.384,E2 -26114.384} C_VEL
LIN {X 0,Y 138.311,Z 233.832,A -85,B 0,C 180,E1 -26118.134,E2 -26118.134} C_VEL
LIN {X 0,Y 139.367,Z 235.086,A -85,B 0,C 180,E1 -26119.613,E2 -26119.613} C_VEL
LIN {X 0,Y 142.653,Z 240.016,A -85,B 0,C 180,E1 -26123.662,E2 -26123.662} C_VEL
LIN {X 0,Y 145.182,Z 243.915,A -85,B 0,C 180,E1 -26126.285,E2 -26126.285} C_VEL
LIN {X 0,Y 148.874,Z 250.035,A -85,B 0,C 180,E1 -26129.632,E2 -26129.632} C_VEL
LIN {X 0,Y 153.554,Z 258.732,A -85,B 0,C 180,E1 -26133.314,E2 -26133.314} C_VEL
LIN {X 0,Y 156.325,Z 265.55,A -85,B 0,C 180,E1 -26135.369,E2 -26135.369} C_VEL
LIN {X 0,Y 156.917,Z 267.299,A -85,B 0,C 180,E1 -26135.808,E2 -26135.808} C_VEL
LIN {X 0,Y 154.398,Z 297.593,A -85,B 0,C 180,E1 -26136.979,E2 -26136.979} C_VEL
LIN {X 0,Y 152.034,Z 311.129,A -85,B 0,C 180,E1 -26137.794,E2 -26137.794} C_VEL
LIN {X 0,Y 149.149,Z 323.103,A -85,B 0,C 180,E1 -26138.972,E2 -26138.972} C_VEL
LIN {X 0,Y 145.442,Z 334.389,A -85,B 0,C 180,E1 -26140.445,E2 -26140.445} C_VEL
LIN {X 0,Y 140.76,Z 346.021,A -85,B 0,C 180,E1 -26142.573,E2 -26142.573} C_VEL
LIN {X 0,Y 135.672,Z 356.475,A -85,B 0,C 180,E1 -26145.109,E2 -26145.109} C_VEL
LIN {X 0,Y 130.843,Z 365.019,A -85,B 0,C 180,E1 -26147.827,E2 -26147.827} C_VEL
LIN {X 0,Y 126.031,Z 372.891,A -85,B 0,C 180,E1 -26151.148,E2 -26151.148} C_VEL
LIN {X 0,Y 120.714,Z 380.583,A -85,B 0,C 180,E1 -26155.416,E2 -26155.416} C_VEL
LIN {X 0,Y 116.795,Z 385.841,A -85,B 0,C 180,E1 -26159.24,E2 -26159.24} C_VEL
LIN {X 0,Y 112.644,Z 390.939,A -85,B 0,C 180,E1 -26164.107,E2 -26164.107} C_VEL
LIN {X 0,Y 109.516,Z 394.896,A -85,B 0,C 180,E1 -26169.334,E2 -26169.334} C_VEL
LIN {X 0,Y 107.203,Z 397.819,A -85,B 0,C 180,E1 -26174.8,E2 -26174.8} C_VEL
LIN {X 0,Y 106.159,Z 399.214,A -85,B 0,C 180,E1 -26178.546,E2 -26178.546} C_VEL
LIN {X 0,Y 105.471,Z 400.207,A -85,B 0,C 180,E1 -26182.343,E2 -26182.343} C_VEL
LIN {X 0,Y 105.126,Z 400.816,A -85,B 0,C 180,E1 -26186.168,E2 -26186.168} C_VEL
LIN {X 0,Y 105.109,Z 401.042,A -85,B 0,C 180,E1 -26190.002,E2 -26190.002} C_VEL
LIN {X 0,Y 105.126,Z 400.844,A -85,B 0,C 180,E1 -26193.835,E2 -26193.835} C_VEL
LIN {X 0,Y 105.472,Z 400.254,A -85,B 0,C 180,E1 -26197.66,E2 -26197.66} C_VEL
LIN {X 0,Y 106.16,Z 399.279,A -85,B 0,C 180,E1 -26201.457,E2 -26201.457} C_VEL
LIN {X 0,Y 107.203,Z 397.912,A -85,B 0,C 180,E1 -26205.204,E2 -26205.204} C_VEL
LIN {X 0,Y 109.498,Z 395.026,A -85,B 0,C 180,E1 -26210.673,E2 -26210.673} C_VEL
LIN {X 0,Y 112.599,Z 391.114,A -85,B 0,C 180,E1 -26215.908,E2 -26215.908} C_VEL
LIN {X 0,Y 116.739,Z 386.067,A -85,B 0,C 180,E1 -26220.78,E2 -26220.78} C_VEL
LIN {X 0,Y 121.518,Z 379.712,A -85,B 0,C 180,E1 -26225.335,E2 -26225.335} C_VEL
LIN {X 0,Y 126.811,Z 371.767,A -85,B 0,C 180,E1 -26229.595,E2 -26229.595} C_VEL
LIN {X 0,Y 131.766,Z 363.668,A -85,B 0,C 180,E1 -26232.848,E2 -26232.848} C_VEL
LIN {X 0,Y 137.251,Z 353.784,A -85,B 0,C 180,E1 -26235.798,E2 -26235.798} C_VEL
LIN {X 0,Y 142.436,Z 342.651,A -85,B 0,C 180,E1 -26238.27,E2 -26238.27} C_VEL
LIN {X 0,Y 146.564,Z 331.741,A -85,B 0,C 180,E1 -26240.106,E2 -26240.106} C_VEL
LIN {X 0,Y 150.274,Z 319.675,A -85,B 0,C 180,E1 -26241.57,E2 -26241.57} C_VEL
LIN {X 0,Y 153.172,Z 306.643,A -85,B 0,C 180,E1 -26242.679,E2 -26242.679} C_VEL
LIN {X 0,Y 154.981,Z 293.928,A -85,B 0,C 180,E1 -26243.355,E2 -26243.355} C_VEL
LIN {X 0,Y 157.111,Z 267.378,A -85,B 0,C 180,E1 -26244.353,E2 -26244.353} C_VEL
LIN {X 0,Y 154.136,Z 259.62,A -85,B 0,C 180,E1 -26246.566,E2 -26246.566} C_VEL
LIN {X 0,Y 149.542,Z 251.042,A -85,B 0,C 180,E1 -26250.14,E2 -26250.14} C_VEL
LIN {X 0,Y 145.696,Z 244.611,A -85,B 0,C 180,E1 -26253.587,E2 -26253.587} C_VEL
LIN {X 0,Y 142.206,Z 239.04,A -85,B 0,C 180,E1 -26257.287,E2 -26257.287} C_VEL
LIN {X 0,Y 139.384,Z 234.966,A -85,B 0,C 180,E1 -26260.868,E2 -26260.868} C_VEL
LIN {X 0,Y 136.5,Z 230.945,A -85,B 0,C 180,E1 -26265.558,E2 -26265.558} C_VEL
LIN {X 0,Y 136.042,Z 229.923,A -85,B 0,C 180,E1 -26266.557,E2 -26266.557} C_VEL
LIN {X 0,Y 133.452,Z 226.804,A -85,B 0,C 180,E1 -26273.954,E2 -26273.954} C_VEL
LIN {X 0,Y 132.988,Z 224.985,A -85,B 0,C 180,E1 -26278.486,E2 -26278.486} C_VEL
LIN {X 0,Y 132.978,Z 224.81,A -85,B 0,C 180,E1 -26280.757,E2 -26280.757} C_VEL
LIN {X 0,Y 133.22,Z 226.2,A -85,B 0,C 180,E1 -26284.539,E2 -26284.539} C_VEL
LIN {X 0,Y 135.892,Z 229.858,A -85,B 0,C 180,E1 -26293.077,E2 -26293.077} C_VEL
LIN {X 0,Y 136.492,Z 230.957,A -85,B 0,C 180,E1 -26294.347,E2 -26294.347} C_VEL
LIN {X 0,Y 138.819,Z 234.293,A -85,B 0,C 180,E1 -26298.255,E2 -26298.255} C_VEL
LIN {X 0,Y 139.977,Z 236.094,A -85,B 0,C 180,E1 -26299.906,E2 -26299.906} C_VEL
LIN {X 0,Y 142.694,Z 239.926,A -85,B 0,C 180,E1 -26303.205,E2 -26303.205} C_VEL
LIN {X 0,Y 145.86,Z 244.913,A -85,B 0,C 180,E1 -26306.492,E2 -26306.492} C_VEL
LIN {X 0,Y 149.678,Z 251.312,A -85,B 0,C 180,E1 -26309.892,E2 -26309.892} C_VEL
LIN {X 0,Y 152.239,Z 256.668,A -85,B 0,C 180,E1 -26311.995,E2 -26311.995} C_VEL
LIN {X 0,Y 156.154,Z 266.719,A -85,B 0,C 180,E1 -26315.018,E2 -26315.018} C_VEL
LIN {X 0,Y 157.043,Z 269.394,A -85,B 0,C 180,E1 -26315.684,E2 -26315.684} C_VEL
LIN {X 0,Y 154.399,Z 299.79,A -85,B 0,C 180,E1 -26316.822,E2 -26316.822} C_VEL
LIN {X 0,Y 151.957,Z 313.718,A -85,B 0,C 180,E1 -26317.696,E2 -26317.696} C_VEL
LIN {X 0,Y 148.856,Z 325.68,A -85,B 0,C 180,E1 -26318.829,E2 -26318.829} C_VEL
LIN {X 0,Y 144.522,Z 338.314,A -85,B 0,C 180,E1 -26320.551,E2 -26320.551} C_VEL
LIN {X 0,Y 139.855,Z 349.557,A -85,B 0,C 180,E1 -26322.698,E2 -26322.698} C_VEL
LIN {X 0,Y 134.731,Z 359.678,A -85,B 0,C 180,E1 -26325.234,E2 -26325.234} C_VEL
LIN {X 0,Y 129.411,Z 368.8,A -85,B 0,C 180,E1 -26328.297,E2 -26328.297} C_VEL
LIN {X 0,Y 123.649,Z 377.693,A -85,B 0,C 180,E1 -26332.338,E2 -26332.338} C_VEL
LIN {X 0,Y 118.669,Z 384.843,A -85,B 0,C 180,E1 -26336.782,E2 -26336.782} C_VEL
LIN {X 0,Y 114.899,Z 389.669,A -85,B 0,C 180,E1 -26340.702,E2 -26340.702} C_VEL
LIN {X 0,Y 111.089,Z 394.357,A -85,B 0,C 180,E1 -26345.717,E2 -26345.717} C_VEL
LIN {X 0,Y 108.284,Z 397.939,A -85,B 0,C 180,E1 -26351.063,E2 -26351.063} C_VEL
LIN {X 0,Y 106.892,Z 399.784,A -85,B 0,C 180,E1 -26354.751,E2 -26354.751} C_VEL
LIN {X 0,Y 105.304,Z 402.155,A -85,B 0,C 180,E1 -26362.328,E2 -26362.328} C_VEL
LIN {X 0,Y 105.046,Z 402.757,A -85,B 0,C 180,E1 -26366.162,E2 -26366.162} C_VEL
LIN {X 0,Y 105.039,Z 402.965,A -85,B 0,C 180,E1 -26369.998,E2 -26369.998} C_VEL
LIN {X 0,Y 105.045,Z 402.739,A -85,B 0,C 180,E1 -26373.834,E2 -26373.834} C_VEL
LIN {X 0,Y 105.304,Z 402.127,A -85,B 0,C 180,E1 -26377.669,E2 -26377.669} C_VEL
LIN {X 0,Y 105.905,Z 401.128,A -85,B 0,C 180,E1 -26381.481,E2 -26381.481} C_VEL
LIN {X 0,Y 106.901,Z 399.727,A -85,B 0,C 180,E1 -26385.244,E2 -26385.244} C_VEL
LIN {X 0,Y 109.096,Z 396.792,A -85,B 0,C 180,E1 -26390.749,E2 -26390.749} C_VEL
LIN {X 0,Y 112.254,Z 392.821,A -85,B 0,C 180,E1 -26395.99,E2 -26395.99} C_VEL
LIN {X 0,Y 117.032,Z 386.714,A -85,B 0,C 180,E1 -26401.696,E2 -26401.696} C_VEL
LIN {X 0,Y 121.732,Z 380.295,A -85,B 0,C 180,E1 -26406.073,E2 -26406.073} C_VEL
LIN {X 0,Y 127.357,Z 371.771,A -85,B 0,C 180,E1 -26410.419,E2 -26410.419} C_VEL
LIN {X 0,Y 132.2,Z 363.87,A -85,B 0,C 180,E1 -26413.37,E2 -26413.37} C_VEL
LIN {X 0,Y 134.187,Z 359.611,A -85,B 0,C 180,E1 -26414.907,E2 -26414.907} C_VEL
LIN {X 0,Y 136.035,Z 352.387,A -85,B 0,C 180,E1 -26417.67,E2 -26417.67} C_VEL
LIN {X 0,Y 137.678,Z 344.694,A -85,B 0,C 180,E1 -26420.197,E2 -26420.197} C_VEL
LIN {X 0,Y 139.26,Z 339.697,A -85,B 0,C 180,E1 -26421.33,E2 -26421.33} C_VEL
LIN {X 0,Y 143.863,Z 326.982,A -85,B 0,C 180,E1 -26423.121,E2 -26423.121} C_VEL
LIN {X 0,Y 147.128,Z 315.249,A -85,B 0,C 180,E1 -26424.293,E2 -26424.293} C_VEL
LIN {X 0,Y 149.654,Z 302.158,A -85,B 0,C 180,E1 -26425.171,E2 -26425.171} C_VEL
LIN {X 0,Y 151.518,Z 284.193,A -85,B 0,C 180,E1 -26425.89,E2 -26425.89} C_VEL
LIN {X 0,Y 152.534,Z 271.537,A -85,B 0,C 180,E1 -26426.37,E2 -26426.37} C_VEL
LIN {X 0,Y 149.47,Z 262.925,A -85,B 0,C 180,E1 -26428.948,E2 -26428.948} C_VEL
LIN {X 0,Y 147.084,Z 257.357,A -85,B 0,C 180,E1 -26431.067,E2 -26431.067} C_VEL
LIN {X 0,Y 143.224,Z 250.455,A -85,B 0,C 180,E1 -26434.767,E2 -26434.767} C_VEL
LIN {X 0,Y 139.681,Z 244.783,A -85,B 0,C 180,E1 -26438.812,E2 -26438.812} C_VEL
LIN {X 0,Y 137.198,Z 240.929,A -85,B 0,C 180,E1 -26442.293,E2 -26442.293} C_VEL
LIN {X 0,Y 134.804,Z 237.147,A -85,B 0,C 180,E1 -26446.624,E2 -26446.624} C_VEL
LIN {X 0,Y 134.045,Z 236.263,A -85,B 0,C 180,E1 -26448.278,E2 -26448.278} C_VEL
LIN {X 0,Y 131.859,Z 231.882,A -85,B 0,C 180,E1 -26457.709,E2 -26457.709} C_VEL
LIN {X 0,Y 131.785,Z 231.637,A -85,B 0,C 180,E1 -26460.764,E2 -26460.764} C_VEL
LIN {X 0,Y 131.967,Z 232.354,A -85,B 0,C 180,E1 -26463.817,E2 -26463.817} C_VEL
LIN {X 0,Y 134.134,Z 236.345,A -85,B 0,C 180,E1 -26472.098,E2 -26472.098} C_VEL
LIN {X 0,Y 134.815,Z 237.133,A -85,B 0,C 180,E1 -26473.568,E2 -26473.568} C_VEL
LIN {X 0,Y 137.212,Z 240.922,A -85,B 0,C 180,E1 -26477.898,E2 -26477.898} C_VEL
LIN {X 0,Y 140.75,Z 246.408,A -85,B 0,C 180,E1 -26482.666,E2 -26482.666} C_VEL
LIN {X 0,Y 143.479,Z 250.889,A -85,B 0,C 180,E1 -26485.671,E2 -26485.671} C_VEL
LIN {X 0,Y 147.645,Z 258.362,A -85,B 0,C 180,E1 -26489.595,E2 -26489.595} C_VEL
LIN {X 0,Y 151.133,Z 265.486,A -85,B 0,C 180,E1 -26492.477,E2 -26492.477} C_VEL
LIN {X 0,Y 152.651,Z 269.68,A -85,B 0,C 180,E1 -26493.715,E2 -26493.715} C_VEL
LIN {X 0,Y 150.292,Z 297.329,A -85,B 0,C 180,E1 -26494.803,E2 -26494.803} C_VEL
LIN {X 0,Y 147.983,Z 310.371,A -85,B 0,C 180,E1 -26495.564,E2 -26495.564} C_VEL
LIN {X 0,Y 144.797,Z 323.175,A -85,B 0,C 180,E1 -26496.792,E2 -26496.792} C_VEL
LIN {X 0,Y 140.951,Z 334.459,A -85,B 0,C 180,E1 -26498.254,E2 -26498.254} C_VEL
LIN {X 0,Y 136.058,Z 346.09,A -85,B 0,C 180,E1 -26500.371,E2 -26500.371} C_VEL
LIN {X 0,Y 130.746,Z 356.543,A -85,B 0,C 180,E1 -26502.917,E2 -26502.917} C_VEL
LIN {X 0,Y 125.669,Z 365.087,A -85,B 0,C 180,E1 -26505.652,E2 -26505.652} C_VEL
LIN {X 0,Y 120.567,Z 372.959,A -85,B 0,C 180,E1 -26509.024,E2 -26509.024} C_VEL
LIN {X 0,Y 114.941,Z 380.65,A -85,B 0,C 180,E1 -26513.408,E2 -26513.408} C_VEL
LIN {X 0,Y 109.172,Z 387.719,A -85,B 0,C 180,E1 -26519.005,E2 -26519.005} C_VEL
LIN {X 0,Y 105.051,Z 392.426,A -85,B 0,C 180,E1 -26524.227,E2 -26524.227} C_VEL
LIN {X 0,Y 101.942,Z 396.026,A -85,B 0,C 180,E1 -26529.839,E2 -26529.839} C_VEL
LIN {X 0,Y 100.365,Z 397.884,A -85,B 0,C 180,E1 -26533.736,E2 -26533.736} C_VEL
LIN {X 0,Y 99.194,Z 399.279,A -85,B 0,C 180,E1 -26537.73,E2 -26537.73} C_VEL
LIN {X 0,Y 98.041,Z 400.881,A -85,B 0,C 180,E1 -26545.891,E2 -26545.891} C_VEL
LIN {X 0,Y 98.01,Z 401.107,A -85,B 0,C 180,E1 -26550.002,E2 -26550.002} C_VEL
LIN {X 0,Y 98.041,Z 400.909,A -85,B 0,C 180,E1 -26554.112,E2 -26554.112} C_VEL
LIN {X 0,Y 99.194,Z 399.344,A -85,B 0,C 180,E1 -26562.273,E2 -26562.273} C_VEL
LIN {X 0,Y 100.364,Z 397.977,A -85,B 0,C 180,E1 -26566.268,E2 -26566.268} C_VEL
LIN {X 0,Y 102.869,Z 395.09,A -85,B 0,C 180,E1 -26572.073,E2 -26572.073} C_VEL
LIN {X 0,Y 106.256,Z 391.178,A -85,B 0,C 180,E1 -26577.582,E2 -26577.582} C_VEL
LIN {X 0,Y 110.695,Z 386.13,A -85,B 0,C 180,E1 -26582.662,E2 -26582.662} C_VEL
LIN {X 0,Y 115.788,Z 379.775,A -85,B 0,C 180,E1 -26587.372,E2 -26587.372} C_VEL
LIN {X 0,Y 121.4,Z 371.83,A -85,B 0,C 180,E1 -26591.741,E2 -26591.741} C_VEL
LIN {X 0,Y 126.659,Z 363.73,A -85,B 0,C 180,E1 -26595.03,E2 -26595.03} C_VEL
LIN {X 0,Y 132.393,Z 353.846,A -85,B 0,C 180,E1 -26598.004,E2 -26598.004} C_VEL
LIN {X 0,Y 137.809,Z 342.712,A -85,B 0,C 180,E1 -26600.475,E2 -26600.475} C_VEL
LIN {X 0,Y 142.129,Z 331.8,A -85,B 0,C 180,E1 -26602.295,E2 -26602.295} C_VEL
LIN {X 0,Y 145.975,Z 319.733,A -85,B 0,C 180,E1 -26603.749,E2 -26603.749} C_VEL
LIN {X 0,Y 148.933,Z 306.921,A -85,B 0,C 180,E1 -26604.838,E2 -26604.838} C_VEL
LIN {X 0,Y 150.84,Z 294.062,A -85,B 0,C 180,E1 -26605.516,E2 -26605.516} C_VEL
LIN {X 0,Y 152.877,Z 269.812,A -85,B 0,C 180,E1 -26606.43,E2 -26606.43} C_VEL
LIN {X 0,Y 150.382,Z 263.5,A -85,B 0,C 180,E1 -26608.453,E2 -26608.453} C_VEL
LIN {X 0,Y 145.863,Z 254.835,A -85,B 0,C 180,E1 -26612.37,E2 -26612.37} C_VEL
LIN {X 0,Y 142.24,Z 248.577,A -85,B 0,C 180,E1 -26616.062,E2 -26616.062} C_VEL
LIN {X 0,Y 139.76,Z 244.739,A -85,B 0,C 180,E1 -26619.005,E2 -26619.005} C_VEL
LIN {X 0,Y 137.309,Z 240.943,A -85,B 0,C 180,E1 -26622.5,E2 -26622.5} C_VEL
LIN {X 0,Y 135.086,Z 237.497,A -85,B 0,C 180,E1 -26626.556,E2 -26626.556} C_VEL
LIN {X 0,Y 134.644,Z 236.684,A -85,B 0,C 180,E1 -26627.566,E2 -26627.566} C_VEL
LIN {X 0,Y 132.108,Z 231.895,A -85,B 0,C 180,E1 -26639.149,E2 -26639.149} C_VEL
LIN {X 0,Y 132.124,Z 232.061,A -85,B 0,C 180,E1 -26641.524,E2 -26641.524} C_VEL
LIN {X 0,Y 134.943,Z 237.169,A -85,B 0,C 180,E1 -26653.027,E2 -26653.027} C_VEL
LIN {X 0,Y 137.127,Z 240.753,A -85,B 0,C 180,E1 -26657.139,E2 -26657.139} C_VEL
LIN {X 0,Y 138.105,Z 242.222,A -85,B 0,C 180,E1 -26658.641,E2 -26658.641} C_VEL
LIN {X 0,Y 140.925,Z 246.524,A -85,B 0,C 180,E1 -26662.35,E2 -26662.35} C_VEL
LIN {X 0,Y 144.58,Z 252.549,A -85,B 0,C 180,E1 -26666.307,E2 -26666.307} C_VEL
LIN {X 0,Y 148.046,Z 259.088,A -85,B 0,C 180,E1 -26669.534,E2 -26669.534} C_VEL
LIN {X 0,Y 151.406,Z 267.758,A -85,B 0,C 180,E1 -26672.46,E2 -26672.46} C_VEL
LIN {X 0,Y 152.767,Z 271.677,A -85,B 0,C 180,E1 -26673.58,E2 -26673.58} C_VEL
LIN {X 0,Y 150.227,Z 300.001,A -85,B 0,C 180,E1 -26674.674,E2 -26674.674} C_VEL
LIN {X 0,Y 147.754,Z 313.571,A -85,B 0,C 180,E1 -26675.516,E2 -26675.516} C_VEL
LIN {X 0,Y 144.525,Z 325.622,A -85,B 0,C 180,E1 -26676.643,E2 -26676.643} C_VEL
LIN {X 0,Y 140.017,Z 338.254,A -85,B 0,C 180,E1 -26678.346,E2 -26678.346} C_VEL
LIN {X 0,Y 135.137,Z 349.496,A -85,B 0,C 180,E1 -26680.483,E2 -26680.483} C_VEL
LIN {X 0,Y 129.775,Z 359.616,A -85,B 0,C 180,E1 -26683.021,E2 -26683.021} C_VEL
LIN {X 0,Y 124.193,Z 368.737,A -85,B 0,C 180,E1 -26686.114,E2 -26686.114} C_VEL
LIN {X 0,Y 117.993,Z 377.764,A -85,B 0,C 180,E1 -26690.296,E2 -26690.296} C_VEL
LIN {X 0,Y 112.78,Z 384.8,A -85,B 0,C 180,E1 -26694.821,E2 -26694.821} C_VEL
LIN {X 0,Y 108.728,Z 389.605,A -85,B 0,C 180,E1 -26698.861,E2 -26698.861} C_VEL
LIN {X 0,Y 104.642,Z 394.293,A -85,B 0,C 180,E1 -26704.115,E2 -26704.115} C_VEL
LIN {X 0,Y 101.554,Z 397.874,A -85,B 0,C 180,E1 -26709.754,E2 -26709.754} C_VEL
LIN {X 0,Y 100.051,Z 399.719,A -85,B 0,C 180,E1 -26713.68,E2 -26713.68} C_VEL
LIN {X 0,Y 98.272,Z 402.09,A -85,B 0,C 180,E1 -26721.775,E2 -26721.775} C_VEL
LIN {X 0,Y 97.953,Z 402.692,A -85,B 0,C 180,E1 -26725.884,E2 -26725.884} C_VEL
LIN {X 0,Y 97.946,Z 402.9,A -85,B 0,C 180,E1 -26729.998,E2 -26729.998} C_VEL
LIN {X 0,Y 97.952,Z 402.674,A -85,B 0,C 180,E1 -26734.113,E2 -26734.113} C_VEL
LIN {X 0,Y 98.272,Z 402.061,A -85,B 0,C 180,E1 -26738.221,E2 -26738.221} C_VEL
LIN {X 0,Y 100.058,Z 399.661,A -85,B 0,C 180,E1 -26746.315,E2 -26746.315} C_VEL
LIN {X 0,Y 102.446,Z 396.725,A -85,B 0,C 180,E1 -26752.165,E2 -26752.165} C_VEL
LIN {X 0,Y 105.903,Z 392.755,A -85,B 0,C 180,E1 -26757.678,E2 -26757.678} C_VEL
LIN {X 0,Y 111.05,Z 386.648,A -85,B 0,C 180,E1 -26763.622,E2 -26763.622} C_VEL
LIN {X 0,Y 116.142,Z 380.103,A -85,B 0,C 180,E1 -26768.22,E2 -26768.22} C_VEL
LIN {X 0,Y 122.039,Z 371.703,A -85,B 0,C 180,E1 -26772.58,E2 -26772.58} C_VEL
LIN {X 0,Y 127.478,Z 363.211,A -85,B 0,C 180,E1 -26775.78,E2 -26775.78} C_VEL
LIN {X 0,Y 133.253,Z 352.717,A -85,B 0,C 180,E1 -26778.723,E2 -26778.723} C_VEL
LIN {X 0,Y 138.183,Z 342.329,A -85,B 0,C 180,E1 -26780.857,E2 -26780.857} C_VEL
LIN {X 0,Y 139.26,Z 339.697,A -85,B 0,C 180,E1 -26781.33,E2 -26781.33} C_VEL
LIN {X 0,Y 140.76,Z 334.59,A -85,B 0,C 180,E1 -26782.381,E2 -26782.381} C_VEL
LIN {X 0,Y 142.279,Z 322.646,A -85,B 0,C 180,E1 -26785.209,E2 -26785.209} C_VEL
LIN {X 0,Y 143.197,Z 315.477,A -85,B 0,C 180,E1 -26786.471,E2 -26786.471} C_VEL
LIN {X 0,Y 143.908,Z 311.737,A -85,B 0,C 180,E1 -26786.849,E2 -26786.849} C_VEL
LIN {X 0,Y 146.26,Z 298.62,A -85,B 0,C 180,E1 -26787.615,E2 -26787.615} C_VEL
LIN {X 0,Y 148.515,Z 274.024,A -85,B 0,C 180,E1 -26788.543,E2 -26788.543} C_VEL
LIN {X 0,Y 145.309,Z 265.006,A -85,B 0,C 180,E1 -26791.569,E2 -26791.569} C_VEL
LIN {X 0,Y 143.173,Z 260.445,A -85,B 0,C 180,E1 -26793.684,E2 -26793.684} C_VEL
LIN {X 0,Y 139.781,Z 254.347,A -85,B 0,C 180,E1 -26797.422,E2 -26797.422} C_VEL
LIN {X 0,Y 137.869,Z 251.158,A -85,B 0,C 180,E1 -26799.874,E2 -26799.874} C_VEL
LIN {X 0,Y 135.631,Z 247.494,A -85,B 0,C 180,E1 -26803.267,E2 -26803.267} C_VEL
LIN {X 0,Y 133.187,Z 243.395,A -85,B 0,C 180,E1 -26808.201,E2 -26808.201} C_VEL
LIN {X 0,Y 130.991,Z 238.956,A -85,B 0,C 180,E1 -26817.694,E2 -26817.694} C_VEL
LIN {X 0,Y 130.918,Z 238.696,A -85,B 0,C 180,E1 -26820.769,E2 -26820.769} C_VEL
LIN {X 0,Y 131.054,Z 239.366,A -85,B 0,C 180,E1 -26823.459,E2 -26823.459} C_VEL
LIN {X 0,Y 132.943,Z 243.213,A -85,B 0,C 180,E1 -26831.413,E2 -26831.413} C_VEL
LIN {X 0,Y 133.525,Z 243.906,A -85,B 0,C 180,E1 -26832.766,E2 -26832.766} C_VEL
LIN {X 0,Y 136.374,Z 248.678,A -85,B 0,C 180,E1 -26838.109,E2 -26838.109} C_VEL
LIN {X 0,Y 138.841,Z 252.727,A -85,B 0,C 180,E1 -26841.58,E2 -26841.58} C_VEL
LIN {X 0,Y 142.027,Z 258.254,A -85,B 0,C 180,E1 -26845.289,E2 -26845.289} C_VEL
LIN {X 0,Y 146.234,Z 266.518,A -85,B 0,C 180,E1 -26849.414,E2 -26849.414} C_VEL
LIN {X 0,Y 148.527,Z 272.011,A -85,B 0,C 180,E1 -26851.455,E2 -26851.455} C_VEL
LIN {X 0,Y 148.64,Z 272.376,A -85,B 0,C 180,E1 -26851.56,E2 -26851.56} C_VEL
LIN {X 0,Y 146.172,Z 298.584,A -85,B 0,C 180,E1 -26852.572,E2 -26852.572} C_VEL
LIN {X 0,Y 143.551,Z 312.318,A -85,B 0,C 180,E1 -26853.403,E2 -26853.403} C_VEL
LIN {X 0,Y 140.341,Z 324.321,A -85,B 0,C 180,E1 -26854.602,E2 -26854.602} C_VEL
LIN {X 0,Y 136.016,Z 336.111,A -85,B 0,C 180,E1 -26856.166,E2 -26856.166} C_VEL
LIN {X 0,Y 130.95,Z 347.449,A -85,B 0,C 180,E1 -26858.291,E2 -26858.291} C_VEL
LIN {X 0,Y 125.412,Z 357.667,A -85,B 0,C 180,E1 -26860.845,E2 -26860.845} C_VEL
LIN {X 0,Y 119.579,Z 366.843,A -85,B 0,C 180,E1 -26863.952,E2 -26863.952} C_VEL
LIN {X 0,Y 113.407,Z 375.553,A -85,B 0,C 180,E1 -26868.045,E2 -26868.045} C_VEL
LIN {X 0,Y 107.451,Z 382.944,A -85,B 0,C 180,E1 -26872.773,E2 -26872.773} C_VEL
LIN {X 0,Y 103.152,Z 387.786,A -85,B 0,C 180,E1 -26876.974,E2 -26876.974} C_VEL
LIN {X 0,Y 98.698,Z 392.492,A -85,B 0,C 180,E1 -26882.432,E2 -26882.432} C_VEL
LIN {X 0,Y 95.296,Z 396.092,A -85,B 0,C 180,E1 -26888.364,E2 -26888.364} C_VEL
LIN {X 0,Y 93.558,Z 397.95,A -85,B 0,C 180,E1 -26892.516,E2 -26892.516} C_VEL
LIN {X 0,Y 92.264,Z 399.345,A -85,B 0,C 180,E1 -26896.792,E2 -26896.792} C_VEL
LIN {X 0,Y 90.952,Z 400.946,A -85,B 0,C 180,E1 -26905.57,E2 -26905.57} C_VEL
LIN {X 0,Y 90.918,Z 401.172,A -85,B 0,C 180,E1 -26910.002,E2 -26910.002} C_VEL
LIN {X 0,Y 90.953,Z 400.974,A -85,B 0,C 180,E1 -26914.434,E2 -26914.434} C_VEL
LIN {X 0,Y 92.265,Z 399.408,A -85,B 0,C 180,E1 -26923.211,E2 -26923.211} C_VEL
LIN {X 0,Y 93.557,Z 398.041,A -85,B 0,C 180,E1 -26927.488,E2 -26927.488} C_VEL
LIN {X 0,Y 96.312,Z 395.154,A -85,B 0,C 180,E1 -26933.663,E2 -26933.663} C_VEL
LIN {X 0,Y 100.018,Z 391.241,A -85,B 0,C 180,E1 -26939.465,E2 -26939.465} C_VEL
LIN {X 0,Y 104.785,Z 386.194,A -85,B 0,C 180,E1 -26944.758,E2 -26944.758} C_VEL
LIN {X 0,Y 110.227,Z 379.838,A -85,B 0,C 180,E1 -26949.613,E2 -26949.613} C_VEL
LIN {X 0,Y 116.198,Z 371.893,A -85,B 0,C 180,E1 -26954.072,E2 -26954.072} C_VEL
LIN {X 0,Y 121.75,Z 363.792,A -85,B 0,C 180,E1 -26957.392,E2 -26957.392} C_VEL
LIN {X 0,Y 127.744,Z 353.908,A -85,B 0,C 180,E1 -26960.375,E2 -26960.375} C_VEL
LIN {X 0,Y 133.395,Z 342.772,A -85,B 0,C 180,E1 -26962.833,E2 -26962.833} C_VEL
LIN {X 0,Y 137.913,Z 331.859,A -85,B 0,C 180,E1 -26964.623,E2 -26964.623} C_VEL
LIN {X 0,Y 141.897,Z 319.79,A -85,B 0,C 180,E1 -26966.059,E2 -26966.059} C_VEL
LIN {X 0,Y 144.868,Z 307.567,A -85,B 0,C 180,E1 -26967.084,E2 -26967.084} C_VEL
LIN {X 0,Y 146.904,Z 294.491,A -85,B 0,C 180,E1 -26967.779,E2 -26967.779} C_VEL
LIN {X 0,Y 148.839,Z 272.514,A -85,B 0,C 180,E1 -26968.607,E2 -26968.607} C_VEL
LIN {X 0,Y 147.222,Z 268.34,A -85,B 0,C 180,E1 -26970.053,E2 -26970.053} C_VEL
LIN {X 0,Y 143.188,Z 260.253,A -85,B 0,C 180,E1 -26973.883,E2 -26973.883} C_VEL
LIN {X 0,Y 140.068,Z 254.55,A -85,B 0,C 180,E1 -26977.36,E2 -26977.36} C_VEL
LIN {X 0,Y 137.827,Z 250.93,A -85,B 0,C 180,E1 -26980.256,E2 -26980.256} C_VEL
LIN {X 0,Y 135.769,Z 247.51,A -85,B 0,C 180,E1 -26983.459,E2 -26983.459} C_VEL
LIN {X 0,Y 133.645,Z 243.848,A -85,B 0,C 180,E1 -26987.761,E2 -26987.761} C_VEL
LIN {X 0,Y 131.238,Z 238.984,A -85,B 0,C 180,E1 -26999.143,E2 -26999.143} C_VEL
LIN {X 0,Y 131.241,Z 238.904,A -85,B 0,C 180,E1 -27000.508,E2 -27000.508} C_VEL
LIN {X 0,Y 133.693,Z 243.976,A -85,B 0,C 180,E1 -27012.283,E2 -27012.283} C_VEL
LIN {X 0,Y 135.706,Z 247.454,A -85,B 0,C 180,E1 -27016.358,E2 -27016.358} C_VEL
LIN {X 0,Y 138.904,Z 252.633,A -85,B 0,C 180,E1 -27021.106,E2 -27021.106} C_VEL
LIN {X 0,Y 142.238,Z 258.427,A -85,B 0,C 180,E1 -27025.029,E2 -27025.029} C_VEL
LIN {X 0,Y 145.217,Z 264.431,A -85,B 0,C 180,E1 -27028.057,E2 -27028.057} C_VEL
LIN {X 0,Y 147.984,Z 272.042,A -85,B 0,C 180,E1 -27030.717,E2 -27030.717} C_VEL
LIN {X 0,Y 148.729,Z 274.166,A -85,B 0,C 180,E1 -27031.39,E2 -27031.39} C_VEL
LIN {X 0,Y 146.281,Z 300.14,A -85,B 0,C 180,E1 -27032.4,E2 -27032.4} C_VEL
LIN {X 0,Y 143.656,Z 313.943,A -85,B 0,C 180,E1 -27033.247,E2 -27033.247} C_VEL
LIN {X 0,Y 140.412,Z 325.563,A -85,B 0,C 180,E1 -27034.323,E2 -27034.323} C_VEL
LIN {X 0,Y 135.732,Z 338.194,A -85,B 0,C 180,E1 -27035.997,E2 -27035.997} C_VEL
LIN {X 0,Y 130.63,Z 349.435,A -85,B 0,C 180,E1 -27038.109,E2 -27038.109} C_VEL
LIN {X 0,Y 125.042,Z 359.554,A -85,B 0,C 180,E1 -27040.644,E2 -27040.644} C_VEL
LIN {X 0,Y 119.168,Z 368.675,A -85,B 0,C 180,E1 -27043.742,E2 -27043.742} C_VEL
LIN {X 0,Y 112.703,Z 377.565,A -85,B 0,C 180,E1 -27047.905,E2 -27047.905} C_VEL
LIN {X 0,Y 107.065,Z 384.716,A -85,B 0,C 180,E1 -27052.612,E2 -27052.612} C_VEL
LIN {X 0,Y 102.686,Z 389.541,A -85,B 0,C 180,E1 -27056.801,E2 -27056.801} C_VEL
LIN {X 0,Y 98.293,Z 394.229,A -85,B 0,C 180,E1 -27062.304,E2 -27062.304} C_VEL
LIN {X 0,Y 94.884,Z 397.81,A -85,B 0,C 180,E1 -27068.262,E2 -27068.262} C_VEL
LIN {X 0,Y 93.222,Z 399.655,A -85,B 0,C 180,E1 -27072.447,E2 -27072.447} C_VEL
LIN {X 0,Y 92.019,Z 401.038,A -85,B 0,C 180,E1 -27076.753,E2 -27076.753} C_VEL
LIN {X 0,Y 91.241,Z 402.026,A -85,B 0,C 180,E1 -27081.136,E2 -27081.136} C_VEL
LIN {X 0,Y 90.883,Z 402.627,A -85,B 0,C 180,E1 -27085.563,E2 -27085.563} C_VEL
LIN {X 0,Y 90.845,Z 402.835,A -85,B 0,C 180,E1 -27089.998,E2 -27089.998} C_VEL
LIN {X 0,Y 90.883,Z 402.609,A -85,B 0,C 180,E1 -27094.433,E2 -27094.433} C_VEL
LIN {X 0,Y 91.24,Z 401.996,A -85,B 0,C 180,E1 -27098.86,E2 -27098.86} C_VEL
LIN {X 0,Y 92.021,Z 400.997,A -85,B 0,C 180,E1 -27103.243,E2 -27103.243} C_VEL
LIN {X 0,Y 93.244,Z 399.596,A -85,B 0,C 180,E1 -27107.545,E2 -27107.545} C_VEL
LIN {X 0,Y 95.878,Z 396.659,A -85,B 0,C 180,E1 -27113.773,E2 -27113.773} C_VEL
LIN {X 0,Y 99.659,Z 392.689,A -85,B 0,C 180,E1 -27119.578,E2 -27119.578} C_VEL
LIN {X 0,Y 105.213,Z 386.581,A -85,B 0,C 180,E1 -27125.763,E2 -27125.763} C_VEL
LIN {X 0,Y 110.723,Z 379.912,A -85,B 0,C 180,E1 -27130.584,E2 -27130.584} C_VEL
LIN {X 0,Y 116.893,Z 371.636,A -85,B 0,C 180,E1 -27134.943,E2 -27134.943} C_VEL
LIN {X 0,Y 122.628,Z 363.143,A -85,B 0,C 180,E1 -27138.16,E2 -27138.16} C_VEL
LIN {X 0,Y 128.685,Z 352.648,A -85,B 0,C 180,E1 -27141.097,E2 -27141.097} C_VEL
LIN {X 0,Y 133.815,Z 342.259,A -85,B 0,C 180,E1 -27143.215,E2 -27143.215} C_VEL
LIN {X 0,Y 138.384,Z 330.851,A -85,B 0,C 180,E1 -27144.973,E2 -27144.973} C_VEL
LIN {X 0,Y 142.058,Z 319.077,A -85,B 0,C 180,E1 -27146.276,E2 -27146.276} C_VEL
LIN {X 0,Y 143.908,Z 311.737,A -85,B 0,C 180,E1 -27146.849,E2 -27146.849} C_VEL
LIN {X 0,Y 144.761,Z 306.072,A -85,B 0,C 180,E1 -27147.42,E2 -27147.42} C_VEL
LIN {X 0,Y 144.638,Z 296.838,A -85,B 0,C 180,E1 -27148.854,E2 -27148.854} C_VEL
LIN {X 0,Y 144.069,Z 287.512,A -85,B 0,C 180,E1 -27150.219,E2 -27150.219} C_VEL
LIN {X 0,Y 144.239,Z 281.693,A -85,B 0,C 180,E1 -27150.66,E2 -27150.66} C_VEL
LIN {X 0,Y 144.657,Z 276.6,A -85,B 0,C 180,E1 -27150.871,E2 -27150.871} C_VEL
LIN {X 0,Y 141.967,Z 268.741,A -85,B 0,C 180,E1 -27153.74,E2 -27153.74} C_VEL
LIN {X 0,Y 138.801,Z 262.412,A -85,B 0,C 180,E1 -27157.331,E2 -27157.331} C_VEL
LIN {X 0,Y 136.068,Z 257.475,A -85,B 0,C 180,E1 -27161.02,E2 -27161.02} C_VEL
LIN {X 0,Y 134.022,Z 253.941,A -85,B 0,C 180,E1 -27164.41,E2 -27164.41} C_VEL
LIN {X 0,Y 132.01,Z 250.252,A -85,B 0,C 180,E1 -27168.873,E2 -27168.873} C_VEL
LIN {X 0,Y 130.082,Z 245.864,A -85,B 0,C 180,E1 -27178.452,E2 -27178.452} C_VEL
LIN {X 0,Y 130.051,Z 245.758,A -85,B 0,C 180,E1 -27180.774,E2 -27180.774} C_VEL
LIN {X 0,Y 130.188,Z 246.65,A -85,B 0,C 180,E1 -27183.676,E2 -27183.676} C_VEL
LIN {X 0,Y 131.889,Z 250.171,A -85,B 0,C 180,E1 -27191.009,E2 -27191.009} C_VEL
LIN {X 0,Y 132.383,Z 250.94,A -85,B 0,C 180,E1 -27192.261,E2 -27192.261} C_VEL
LIN {X 0,Y 134.81,Z 255.255,A -85,B 0,C 180,E1 -27197.15,E2 -27197.15} C_VEL
LIN {X 0,Y 137.171,Z 259.378,A -85,B 0,C 180,E1 -27200.723,E2 -27200.723} C_VEL
LIN {X 0,Y 140.026,Z 264.749,A -85,B 0,C 180,E1 -27204.298,E2 -27204.298} C_VEL
LIN {X 0,Y 143.645,Z 272.366,A -85,B 0,C 180,E1 -27208.135,E2 -27208.135} C_VEL
LIN {X 0,Y 144.827,Z 275.154,A -85,B 0,C 180,E1 -27209.279,E2 -27209.279} C_VEL
LIN {X 0,Y 142.539,Z 298.303,A -85,B 0,C 180,E1 -27210.154,E2 -27210.154} C_VEL
LIN {X 0,Y 139.895,Z 311.853,A -85,B 0,C 180,E1 -27210.935,E2 -27210.935} C_VEL
LIN {X 0,Y 136.443,Z 324.392,A -85,B 0,C 180,E1 -27212.153,E2 -27212.153} C_VEL
LIN {X 0,Y 131.961,Z 336.181,A -85,B 0,C 180,E1 -27213.683,E2 -27213.683} C_VEL
LIN {X 0,Y 126.667,Z 347.518,A -85,B 0,C 180,E1 -27215.766,E2 -27215.766} C_VEL
LIN {X 0,Y 120.891,Z 357.735,A -85,B 0,C 180,E1 -27218.3,E2 -27218.3} C_VEL
LIN {X 0,Y 114.75,Z 366.91,A -85,B 0,C 180,E1 -27221.391,E2 -27221.391} C_VEL
LIN {X 0,Y 109.131,Z 374.478,A -85,B 0,C 180,E1 -27224.899,E2 -27224.899} C_VEL
LIN {X 0,Y 102.862,Z 381.898,A -85,B 0,C 180,E1 -27229.531,E2 -27229.531} C_VEL
LIN {X 0,Y 97.28,Z 387.852,A -85,B 0,C 180,E1 -27234.696,E2 -27234.696} C_VEL
LIN {X 0,Y 92.461,Z 392.558,A -85,B 0,C 180,E1 -27240.395,E2 -27240.395} C_VEL
LIN {X 0,Y 88.728,Z 396.158,A -85,B 0,C 180,E1 -27246.672,E2 -27246.672} C_VEL
LIN {X 0,Y 86.794,Z 398.016,A -85,B 0,C 180,E1 -27251.104,E2 -27251.104} C_VEL
LIN {X 0,Y 85.349,Z 399.41,A -85,B 0,C 180,E1 -27255.701,E2 -27255.701} C_VEL
LIN {X 0,Y 84.391,Z 400.403,A -85,B 0,C 180,E1 -27260.415,E2 -27260.415} C_VEL
LIN {X 0,Y 83.887,Z 401.011,A -85,B 0,C 180,E1 -27265.196,E2 -27265.196} C_VEL
LIN {X 0,Y 83.818,Z 401.237,A -85,B 0,C 180,E1 -27270.002,E2 -27270.002} C_VEL
LIN {X 0,Y 83.888,Z 401.039,A -85,B 0,C 180,E1 -27274.808,E2 -27274.808} C_VEL
LIN {X 0,Y 84.392,Z 400.448,A -85,B 0,C 180,E1 -27279.59,E2 -27279.59} C_VEL
LIN {X 0,Y 86.792,Z 398.105,A -85,B 0,C 180,E1 -27288.901,E2 -27288.901} C_VEL
LIN {X 0,Y 89.818,Z 395.219,A -85,B 0,C 180,E1 -27295.492,E2 -27295.492} C_VEL
LIN {X 0,Y 93.904,Z 391.305,A -85,B 0,C 180,E1 -27301.595,E2 -27301.595} C_VEL
LIN {X 0,Y 99.03,Z 386.257,A -85,B 0,C 180,E1 -27307.103,E2 -27307.103} C_VEL
LIN {X 0,Y 104.845,Z 379.901,A -85,B 0,C 180,E1 -27312.093,E2 -27312.093} C_VEL
LIN {X 0,Y 111.187,Z 371.955,A -85,B 0,C 180,E1 -27316.628,E2 -27316.628} C_VEL
LIN {X 0,Y 117.057,Z 363.854,A -85,B 0,C 180,E1 -27319.952,E2 -27319.952} C_VEL
LIN {X 0,Y 123.343,Z 353.969,A -85,B 0,C 180,E1 -27322.913,E2 -27322.913} C_VEL
LIN {X 0,Y 129.239,Z 342.832,A -85,B 0,C 180,E1 -27325.336,E2 -27325.336} C_VEL
LIN {X 0,Y 133.937,Z 331.918,A -85,B 0,C 180,E1 -27327.094,E2 -27327.094} C_VEL
LIN {X 0,Y 138.069,Z 319.848,A -85,B 0,C 180,E1 -27328.497,E2 -27328.497} C_VEL
LIN {X 0,Y 141.258,Z 307.049,A -85,B 0,C 180,E1 -27329.532,E2 -27329.532} C_VEL
LIN {X 0,Y 143.346,Z 293.409,A -85,B 0,C 180,E1 -27330.243,E2 -27330.243} C_VEL
LIN {X 0,Y 145.05,Z 275.344,A -85,B 0,C 180,E1 -27330.874,E2 -27330.874} C_VEL
LIN {X 0,Y 141.989,Z 268.501,A -85,B 0,C 180,E1 -27333.942,E2 -27333.942} C_VEL
LIN {X 0,Y 138.892,Z 262.322,A -85,B 0,C 180,E1 -27337.501,E2 -27337.501} C_VEL
LIN {X 0,Y 136.2,Z 257.474,A -85,B 0,C 180,E1 -27341.185,E2 -27341.185} C_VEL
LIN {X 0,Y 134.252,Z 254.069,A -85,B 0,C 180,E1 -27344.463,E2 -27344.463} C_VEL
LIN {X 0,Y 132.278,Z 250.426,A -85,B 0,C 180,E1 -27348.895,E2 -27348.895} C_VEL
LIN {X 0,Y 130.378,Z 245.877,A -85,B 0,C 180,E1 -27360,E2 -27360} C_VEL
LIN {X 0,Y 132.446,Z 250.765,A -85,B 0,C 180,E1 -27371.478,E2 -27371.478} C_VEL
LIN {X 0,Y 134.814,Z 255.025,A -85,B 0,C 180,E1 -27376.469,E2 -27376.469} C_VEL
LIN {X 0,Y 137.293,Z 259.375,A -85,B 0,C 180,E1 -27380.312,E2 -27380.312} C_VEL
LIN {X 0,Y 140.309,Z 265.056,A -85,B 0,C 180,E1 -27384.113,E2 -27384.113} C_VEL
LIN {X 0,Y 142.586,Z 270.023,A -85,B 0,C 180,E1 -27386.63,E2 -27386.63} C_VEL
LIN {X 0,Y 144.902,Z 276.919,A -85,B 0,C 180,E1 -27389.094,E2 -27389.094} C_VEL
LIN {X 0,Y 142.649,Z 299.751,A -85,B 0,C 180,E1 -27389.97,E2 -27389.97} C_VEL
LIN {X 0,Y 139.985,Z 313.426,A -85,B 0,C 180,E1 -27390.773,E2 -27390.773} C_VEL
LIN {X 0,Y 136.545,Z 325.505,A -85,B 0,C 180,E1 -27391.869,E2 -27391.869} C_VEL
LIN {X 0,Y 131.688,Z 338.134,A -85,B 0,C 180,E1 -27393.5,E2 -27393.5} C_VEL
LIN {X 0,Y 126.359,Z 349.374,A -85,B 0,C 180,E1 -27395.567,E2 -27395.567} C_VEL
LIN {X 0,Y 120.537,Z 359.492,A -85,B 0,C 180,E1 -27398.082,E2 -27398.082} C_VEL
LIN {X 0,Y 114.366,Z 368.612,A -85,B 0,C 180,E1 -27401.167,E2 -27401.167} C_VEL
LIN {X 0,Y 107.525,Z 377.502,A -85,B 0,C 180,E1 -27405.36,E2 -27405.36} C_VEL
LIN {X 0,Y 101.773,Z 384.328,A -85,B 0,C 180,E1 -27409.916,E2 -27409.916} C_VEL
LIN {X 0,Y 96.798,Z 389.478,A -85,B 0,C 180,E1 -27414.489,E2 -27414.489} C_VEL
LIN {X 0,Y 92.059,Z 394.166,A -85,B 0,C 180,E1 -27420.248,E2 -27420.248} C_VEL
LIN {X 0,Y 88.29,Z 397.745,A -85,B 0,C 180,E1 -27426.545,E2 -27426.545} C_VEL
LIN {X 0,Y 86.444,Z 399.59,A -85,B 0,C 180,E1 -27431.02,E2 -27431.02} C_VEL
LIN {X 0,Y 85.096,Z 400.973,A -85,B 0,C 180,E1 -27435.653,E2 -27435.653} C_VEL
LIN {X 0,Y 84.217,Z 401.961,A -85,B 0,C 180,E1 -27440.39,E2 -27440.39} C_VEL
LIN {X 0,Y 83.802,Z 402.563,A -85,B 0,C 180,E1 -27445.187,E2 -27445.187} C_VEL
LIN {X 0,Y 83.767,Z 402.77,A -85,B 0,C 180,E1 -27449.998,E2 -27449.998} C_VEL
LIN {X 0,Y 83.801,Z 402.544,A -85,B 0,C 180,E1 -27454.809,E2 -27454.809} C_VEL
LIN {X 0,Y 84.217,Z 401.931,A -85,B 0,C 180,E1 -27459.605,E2 -27459.605} C_VEL
LIN {X 0,Y 85.099,Z 400.931,A -85,B 0,C 180,E1 -27464.342,E2 -27464.342} C_VEL
LIN {X 0,Y 86.462,Z 399.53,A -85,B 0,C 180,E1 -27468.971,E2 -27468.971} C_VEL
LIN {X 0,Y 89.405,Z 396.593,A -85,B 0,C 180,E1 -27475.614,E2 -27475.614} C_VEL
LIN {X 0,Y 93.542,Z 392.623,A -85,B 0,C 180,E1 -27481.728,E2 -27481.728} C_VEL
LIN {X 0,Y 99.542,Z 386.515,A -85,B 0,C 180,E1 -27488.151,E2 -27488.151} C_VEL
LIN {X 0,Y 105.42,Z 379.845,A -85,B 0,C 180,E1 -27493.101,E2 -27493.101} C_VEL
LIN {X 0,Y 111.979,Z 371.569,A -85,B 0,C 180,E1 -27497.511,E2 -27497.511} C_VEL
LIN {X 0,Y 118.005,Z 363.075,A -85,B 0,C 180,E1 -27500.732,E2 -27500.732} C_VEL
LIN {X 0,Y 124.354,Z 352.58,A -85,B 0,C 180,E1 -27503.64,E2 -27503.64} C_VEL
LIN {X 0,Y 129.685,Z 342.19,A -85,B 0,C 180,E1 -27505.731,E2 -27505.731} C_VEL
LIN {X 0,Y 134.435,Z 330.781,A -85,B 0,C 180,E1 -27507.452,E2 -27507.452} C_VEL
LIN {X 0,Y 138.246,Z 319.004,A -85,B 0,C 180,E1 -27508.721,E2 -27508.721} C_VEL
LIN {X 0,Y 141.461,Z 305.351,A -85,B 0,C 180,E1 -27509.686,E2 -27509.686} C_VEL
LIN {X 0,Y 143.298,Z 292.21,A -85,B 0,C 180,E1 -27510.278,E2 -27510.278} C_VEL
LIN {X 0,Y 144.239,Z 281.693,A -85,B 0,C 180,E1 -27510.66,E2 -27510.66} C_VEL
LIN {X 0,Y 144.194,Z 279.055,A -85,B 0,C 180,E1 -27510.954,E2 -27510.954} C_VEL
LIN {X 0,Y 143.492,Z 276.038,A -85,B 0,C 180,E1 -27511.772,E2 -27511.772} C_VEL
LIN {X 0,Y 142.017,Z 273.097,A -85,B 0,C 180,E1 -27513.218,E2 -27513.218} C_VEL
LIN {X 0,Y 140.633,Z 271.382,A -85,B 0,C 180,E1 -27514.551,E2 -27514.551} C_VEL
LIN {X 0,Y 135.515,Z 266,A -85,B 0,C 180,E1 -27520.353,E2 -27520.353} C_VEL
LIN {X 0,Y 134.983,Z 264.936,A -85,B 0,C 180,E1 -27521.163,E2 -27521.163} C_VEL
LIN {X 0,Y 132.553,Z 260.515,A -85,B 0,C 180,E1 -27525.413,E2 -27525.413} C_VEL
LIN {X 0,Y 130.745,Z 257.012,A -85,B 0,C 180,E1 -27529.841,E2 -27529.841} C_VEL
LIN {X 0,Y 129.213,Z 252.945,A -85,B 0,C 180,E1 -27538.442,E2 -27538.442} C_VEL
LIN {X 0,Y 129.185,Z 252.816,A -85,B 0,C 180,E1 -27540.779,E2 -27540.779} C_VEL
LIN {X 0,Y 129.273,Z 253.69,A -85,B 0,C 180,E1 -27543.312,E2 -27543.312} C_VEL
LIN {X 0,Y 131.099,Z 257.627,A -85,B 0,C 180,E1 -27551.326,E2 -27551.326} C_VEL
LIN {X 0,Y 133.335,Z 261.92,A -85,B 0,C 180,E1 -27556.261,E2 -27556.261} C_VEL
LIN {X 0,Y 135.441,Z 265.863,A -85,B 0,C 180,E1 -27559.712,E2 -27559.712} C_VEL
LIN {X 0,Y 137.876,Z 270.828,A -85,B 0,C 180,E1 -27563.035,E2 -27563.035} C_VEL
LIN {X 0,Y 140.924,Z 277.669,A -85,B 0,C 180,E1 -27566.582,E2 -27566.582} C_VEL
LIN {X 0,Y 141.206,Z 278.334,A -85,B 0,C 180,E1 -27566.884,E2 -27566.884} C_VEL
LIN {X 0,Y 138.997,Z 299.066,A -85,B 0,C 180,E1 -27567.654,E2 -27567.654} C_VEL
LIN {X 0,Y 136.209,Z 312.725,A -85,B 0,C 180,E1 -27568.445,E2 -27568.445} C_VEL
LIN {X 0,Y 132.442,Z 325.458,A -85,B 0,C 180,E1 -27569.67,E2 -27569.67} C_VEL
LIN {X 0,Y 127.474,Z 337.832,A -85,B 0,C 180,E1 -27571.294,E2 -27571.294} C_VEL
LIN {X 0,Y 121.97,Z 348.863,A -85,B 0,C 180,E1 -27573.337,E2 -27573.337} C_VEL
LIN {X 0,Y 116.622,Z 357.803,A -85,B 0,C 180,E1 -27575.56,E2 -27575.56} C_VEL
LIN {X 0,Y 110.181,Z 366.978,A -85,B 0,C 180,E1 -27578.617,E2 -27578.617} C_VEL
LIN {X 0,Y 103.312,Z 375.62,A -85,B 0,C 180,E1 -27582.715,E2 -27582.715} C_VEL
LIN {X 0,Y 96.5,Z 383.078,A -85,B 0,C 180,E1 -27587.653,E2 -27587.653} C_VEL
LIN {X 0,Y 91.584,Z 387.919,A -85,B 0,C 180,E1 -27592.131,E2 -27592.131} C_VEL
LIN {X 0,Y 86.336,Z 392.625,A -85,B 0,C 180,E1 -27598.057,E2 -27598.057} C_VEL
LIN {X 0,Y 82.251,Z 396.223,A -85,B 0,C 180,E1 -27604.711,E2 -27604.711} C_VEL
LIN {X 0,Y 80.101,Z 398.081,A -85,B 0,C 180,E1 -27609.457,E2 -27609.457} C_VEL
LIN {X 0,Y 78.482,Z 399.476,A -85,B 0,C 180,E1 -27614.419,E2 -27614.419} C_VEL
LIN {X 0,Y 77.394,Z 400.468,A -85,B 0,C 180,E1 -27619.539,E2 -27619.539} C_VEL
LIN {X 0,Y 76.812,Z 401.076,A -85,B 0,C 180,E1 -27624.753,E2 -27624.753} C_VEL
LIN {X 0,Y 76.74,Z 401.302,A -85,B 0,C 180,E1 -27630.002,E2 -27630.002} C_VEL
LIN {X 0,Y 76.812,Z 401.103,A -85,B 0,C 180,E1 -27635.252,E2 -27635.252} C_VEL
LIN {X 0,Y 77.394,Z 400.512,A -85,B 0,C 180,E1 -27640.466,E2 -27640.466} C_VEL
LIN {X 0,Y 80.099,Z 398.17,A -85,B 0,C 180,E1 -27650.548,E2 -27650.548} C_VEL
LIN {X 0,Y 83.44,Z 395.283,A -85,B 0,C 180,E1 -27657.599,E2 -27657.599} C_VEL
LIN {X 0,Y 87.937,Z 391.369,A -85,B 0,C 180,E1 -27664.019,E2 -27664.019} C_VEL
LIN {X 0,Y 93.446,Z 386.321,A -85,B 0,C 180,E1 -27669.739,E2 -27669.739} C_VEL
LIN {X 0,Y 99.686,Z 379.964,A -85,B 0,C 180,E1 -27674.831,E2 -27674.831} C_VEL
LIN {X 0,Y 106.434,Z 372.018,A -85,B 0,C 180,E1 -27679.409,E2 -27679.409} C_VEL
LIN {X 0,Y 112.618,Z 363.916,A -85,B 0,C 180,E1 -27682.72,E2 -27682.72} C_VEL
LIN {X 0,Y 119.196,Z 354.03,A -85,B 0,C 180,E1 -27685.636,E2 -27685.636} C_VEL
LIN {X 0,Y 125.343,Z 342.893,A -85,B 0,C 180,E1 -27688.002,E2 -27688.002} C_VEL
LIN {X 0,Y 130.222,Z 331.977,A -85,B 0,C 180,E1 -27689.713,E2 -27689.713} C_VEL
LIN {X 0,Y 134.506,Z 319.905,A -85,B 0,C 180,E1 -27691.068,E2 -27691.068} C_VEL
LIN {X 0,Y 137.789,Z 307.103,A -85,B 0,C 180,E1 -27692.081,E2 -27692.081} C_VEL
LIN {X 0,Y 139.956,Z 293.554,A -85,B 0,C 180,E1 -27692.756,E2 -27692.756} C_VEL
LIN {X 0,Y 141.399,Z 278.384,A -85,B 0,C 180,E1 -27693.317,E2 -27693.317} C_VEL
LIN {X 0,Y 138.188,Z 271.158,A -85,B 0,C 180,E1 -27697.034,E2 -27697.034} C_VEL
LIN {X 0,Y 135.765,Z 266.208,A -85,B 0,C 180,E1 -27700.337,E2 -27700.337} C_VEL
LIN {X 0,Y 134.248,Z 263.435,A -85,B 0,C 180,E1 -27702.727,E2 -27702.727} C_VEL
LIN {X 0,Y 132.758,Z 260.583,A -85,B 0,C 180,E1 -27705.534,E2 -27705.534} C_VEL
LIN {X 0,Y 130.986,Z 257.138,A -85,B 0,C 180,E1 -27709.957,E2 -27709.957} C_VEL
LIN {X 0,Y 129.509,Z 252.954,A -85,B 0,C 180,E1 -27720,E2 -27720} C_VEL
LIN {X 0,Y 131.271,Z 257.687,A -85,B 0,C 180,E1 -27730.8,E2 -27730.8} C_VEL
LIN {X 0,Y 133.456,Z 261.922,A -85,B 0,C 180,E1 -27735.767,E2 -27735.767} C_VEL
LIN {X 0,Y 135.485,Z 265.696,A -85,B 0,C 180,E1 -27739.163,E2 -27739.163} C_VEL
LIN {X 0,Y 137.938,Z 270.619,A -85,B 0,C 180,E1 -27742.564,E2 -27742.564} C_VEL
LIN {X 0,Y 140.02,Z 275.471,A -85,B 0,C 180,E1 -27745.109,E2 -27745.109} C_VEL
LIN {X 0,Y 141.333,Z 279.639,A -85,B 0,C 180,E1 -27746.685,E2 -27746.685} C_VEL
LIN {X 0,Y 139.146,Z 300.292,A -85,B 0,C 180,E1 -27747.467,E2 -27747.467} C_VEL
LIN {X 0,Y 136.4,Z 313.76,A -85,B 0,C 180,E1 -27748.242,E2 -27748.242} C_VEL
LIN {X 0,Y 132.942,Z 325.447,A -85,B 0,C 180,E1 -27749.276,E2 -27749.276} C_VEL
LIN {X 0,Y 127.901,Z 338.074,A -85,B 0,C 180,E1 -27750.843,E2 -27750.843} C_VEL
LIN {X 0,Y 122.355,Z 349.313,A -85,B 0,C 180,E1 -27752.854,E2 -27752.854} C_VEL
LIN {X 0,Y 116.281,Z 359.43,A -85,B 0,C 180,E1 -27755.319,E2 -27755.319} C_VEL
LIN {X 0,Y 109.824,Z 368.55,A -85,B 0,C 180,E1 -27758.378,E2 -27758.378} C_VEL
LIN {X 0,Y 102.567,Z 377.439,A -85,B 0,C 180,E1 -27762.556,E2 -27762.556} C_VEL
LIN {X 0,Y 96.19,Z 384.516,A -85,B 0,C 180,E1 -27767.383,E2 -27767.383} C_VEL
LIN {X 0,Y 91.094,Z 389.414,A -85,B 0,C 180,E1 -27771.886,E2 -27771.886} C_VEL
LIN {X 0,Y 85.951,Z 394.102,A -85,B 0,C 180,E1 -27777.892,E2 -27777.892} C_VEL
LIN {X 0,Y 81.792,Z 397.681,A -85,B 0,C 180,E1 -27784.554,E2 -27784.554} C_VEL
LIN {X 0,Y 79.736,Z 399.525,A -85,B 0,C 180,E1 -27789.354,E2 -27789.354} C_VEL
LIN {X 0,Y 78.22,Z 400.908,A -85,B 0,C 180,E1 -27794.361,E2 -27794.361} C_VEL
LIN {X 0,Y 77.223,Z 401.896,A -85,B 0,C 180,E1 -27799.511,E2 -27799.511} C_VEL
LIN {X 0,Y 76.741,Z 402.498,A -85,B 0,C 180,E1 -27804.743,E2 -27804.743} C_VEL
LIN {X 0,Y 76.679,Z 402.705,A -85,B 0,C 180,E1 -27809.998,E2 -27809.998} C_VEL
LIN {X 0,Y 76.74,Z 402.479,A -85,B 0,C 180,E1 -27815.252,E2 -27815.252} C_VEL
LIN {X 0,Y 77.223,Z 401.865,A -85,B 0,C 180,E1 -27820.485,E2 -27820.485} C_VEL
LIN {X 0,Y 78.224,Z 400.866,A -85,B 0,C 180,E1 -27825.634,E2 -27825.634} C_VEL
LIN {X 0,Y 79.751,Z 399.464,A -85,B 0,C 180,E1 -27830.637,E2 -27830.637} C_VEL
LIN {X 0,Y 83.046,Z 396.527,A -85,B 0,C 180,E1 -27837.736,E2 -27837.736} C_VEL
LIN {X 0,Y 87.577,Z 392.556,A -85,B 0,C 180,E1 -27844.173,E2 -27844.173} C_VEL
LIN {X 0,Y 94.063,Z 386.448,A -85,B 0,C 180,E1 -27850.822,E2 -27850.822} C_VEL
LIN {X 0,Y 100.333,Z 379.777,A -85,B 0,C 180,E1 -27855.884,E2 -27855.884} C_VEL
LIN {X 0,Y 107.299,Z 371.501,A -85,B 0,C 180,E1 -27860.315,E2 -27860.315} C_VEL
LIN {X 0,Y 113.63,Z 363.007,A -85,B 0,C 180,E1 -27863.514,E2 -27863.514} C_VEL
LIN {X 0,Y 120.283,Z 352.511,A -85,B 0,C 180,E1 -27866.363,E2 -27866.363} C_VEL
LIN {X 0,Y 125.825,Z 342.12,A -85,B 0,C 180,E1 -27868.402,E2 -27868.402} C_VEL
LIN {X 0,Y 130.754,Z 330.71,A -85,B 0,C 180,E1 -27870.074,E2 -27870.074} C_VEL
LIN {X 0,Y 134.702,Z 318.931,A -85,B 0,C 180,E1 -27871.299,E2 -27871.299} C_VEL
LIN {X 0,Y 137.968,Z 305.545,A -85,B 0,C 180,E1 -27872.209,E2 -27872.209} C_VEL
LIN {X 0,Y 139.906,Z 292.242,A -85,B 0,C 180,E1 -27872.797,E2 -27872.797} C_VEL
LIN {X 0,Y 141.067,Z 279.361,A -85,B 0,C 180,E1 -27873.288,E2 -27873.288} C_VEL
LIN {X 0,Y 139.143,Z 273.527,A -85,B 0,C 180,E1 -27875.604,E2 -27875.604} C_VEL
LIN {X 0,Y 136.172,Z 267.231,A -85,B 0,C 180,E1 -27879.415,E2 -27879.415} C_VEL
LIN {X 0,Y 134.983,Z 264.936,A -85,B 0,C 180,E1 -27881.163,E2 -27881.163} C_VEL
LIN {X 0,Y 134.048,Z 263.367,A -85,B 0,C 180,E1 -27882.638,E2 -27882.638} C_VEL
LIN {X 0,Y 132.546,Z 262.302,A -85,B 0,C 180,E1 -27885.054,E2 -27885.054} C_VEL
LIN {X 0,Y 128.995,Z 262.497,A -85,B 0,C 180,E1 -27892.918,E2 -27892.918} C_VEL
LIN {X 0,Y 128.617,Z 261.976,A -85,B 0,C 180,E1 -27894.709,E2 -27894.709} C_VEL
LIN {X 0,Y 128.323,Z 259.875,A -85,B 0,C 180,E1 -27899.216,E2 -27899.216} C_VEL
LIN {X 0,Y 128.332,Z 260.038,A -85,B 0,C 180,E1 -27901.569,E2 -27901.569} C_VEL
LIN {X 0,Y 129.96,Z 264.578,A -85,B 0,C 180,E1 -27910.714,E2 -27910.714} C_VEL
LIN {X 0,Y 131.848,Z 268.479,A -85,B 0,C 180,E1 -27915.259,E2 -27915.259} C_VEL
LIN {X 0,Y 133.698,Z 272.232,A -85,B 0,C 180,E1 -27918.584,E2 -27918.584} C_VEL
LIN {X 0,Y 136.263,Z 277.93,A -85,B 0,C 180,E1 -27922.365,E2 -27922.365} C_VEL
LIN {X 0,Y 137.815,Z 281.765,A -85,B 0,C 180,E1 -27924.371,E2 -27924.371} C_VEL
LIN {X 0,Y 135.823,Z 299.356,A -85,B 0,C 180,E1 -27925.02,E2 -27925.02} C_VEL
LIN {X 0,Y 132.979,Z 312.785,A -85,B 0,C 180,E1 -27925.754,E2 -27925.754} C_VEL
LIN {X 0,Y 129.082,Z 325.529,A -85,B 0,C 180,E1 -27926.936,E2 -27926.936} C_VEL
LIN {X 0,Y 123.939,Z 337.902,A -85,B 0,C 180,E1 -27928.492,E2 -27928.492} C_VEL
LIN {X 0,Y 118.22,Z 348.932,A -85,B 0,C 180,E1 -27930.463,E2 -27930.463} C_VEL
LIN {X 0,Y 112.636,Z 357.872,A -85,B 0,C 180,E1 -27932.617,E2 -27932.617} C_VEL
LIN {X 0,Y 105.886,Z 367.046,A -85,B 0,C 180,E1 -27935.608,E2 -27935.608} C_VEL
LIN {X 0,Y 98.684,Z 375.618,A -85,B 0,C 180,E1 -27939.637,E2 -27939.637} C_VEL
LIN {X 0,Y 91.378,Z 383.144,A -85,B 0,C 180,E1 -27944.653,E2 -27944.653} C_VEL
LIN {X 0,Y 86.082,Z 387.985,A -85,B 0,C 180,E1 -27949.225,E2 -27949.225} C_VEL
LIN {X 0,Y 80.384,Z 392.691,A -85,B 0,C 180,E1 -27955.372,E2 -27955.372} C_VEL
LIN {X 0,Y 75.871,Z 396.289,A -85,B 0,C 180,E1 -27962.412,E2 -27962.412} C_VEL
LIN {X 0,Y 73.493,Z 398.147,A -85,B 0,C 180,E1 -27967.514,E2 -27967.514} C_VEL
LIN {X 0,Y 71.671,Z 399.541,A -85,B 0,C 180,E1 -27972.895,E2 -27972.895} C_VEL
LIN {X 0,Y 69.758,Z 401.141,A -85,B 0,C 180,E1 -27984.22,E2 -27984.22} C_VEL
LIN {X 0,Y 69.652,Z 401.366,A -85,B 0,C 180,E1 -27990.002,E2 -27990.002} C_VEL
LIN {X 0,Y 69.759,Z 401.168,A -85,B 0,C 180,E1 -27995.785,E2 -27995.785} C_VEL
LIN {X 0,Y 71.671,Z 399.602,A -85,B 0,C 180,E1 -28007.11,E2 -28007.11} C_VEL
LIN {X 0,Y 73.491,Z 398.234,A -85,B 0,C 180,E1 -28012.492,E2 -28012.492} C_VEL
LIN {X 0,Y 77.2,Z 395.348,A -85,B 0,C 180,E1 -28020.048,E2 -28020.048} C_VEL
LIN {X 0,Y 82.127,Z 391.433,A -85,B 0,C 180,E1 -28026.801,E2 -28026.801} C_VEL
LIN {X 0,Y 88.088,Z 386.385,A -85,B 0,C 180,E1 -28032.702,E2 -28032.702} C_VEL
LIN {X 0,Y 94.784,Z 380.027,A -85,B 0,C 180,E1 -28037.858,E2 -28037.858} C_VEL
LIN {X 0,Y 101.935,Z 372.081,A -85,B 0,C 180,E1 -28042.456,E2 -28042.456} C_VEL
LIN {X 0,Y 108.47,Z 363.978,A -85,B 0,C 180,E1 -28045.701,E2 -28045.701} C_VEL
LIN {X 0,Y 115.34,Z 354.092,A -85,B 0,C 180,E1 -28048.547,E2 -28048.547} C_VEL
LIN {X 0,Y 121.736,Z 342.953,A -85,B 0,C 180,E1 -28050.832,E2 -28050.832} C_VEL
LIN {X 0,Y 126.797,Z 332.036,A -85,B 0,C 180,E1 -28052.479,E2 -28052.479} C_VEL
LIN {X 0,Y 131.229,Z 319.963,A -85,B 0,C 180,E1 -28053.773,E2 -28053.773} C_VEL
LIN {X 0,Y 134.627,Z 307.128,A -85,B 0,C 180,E1 -28054.744,E2 -28054.744} C_VEL
LIN {X 0,Y 136.846,Z 293.6,A -85,B 0,C 180,E1 -28055.405,E2 -28055.405} C_VEL
LIN {X 0,Y 138.072,Z 281.946,A -85,B 0,C 180,E1 -28055.77,E2 -28055.77} C_VEL
LIN {X 0,Y 135.375,Z 275.484,A -85,B 0,C 180,E1 -28059.387,E2 -28059.387} C_VEL
LIN {X 0,Y 133.058,Z 270.561,A -85,B 0,C 180,E1 -28063.112,E2 -28063.112} C_VEL
LIN {X 0,Y 131.301,Z 267.067,A -85,B 0,C 180,E1 -28066.654,E2 -28066.654} C_VEL
LIN {X 0,Y 129.864,Z 263.976,A -85,B 0,C 180,E1 -28070.656,E2 -28070.656} C_VEL
LIN {X 0,Y 128.64,Z 260.036,A -85,B 0,C 180,E1 -28080,E2 -28080} C_VEL
LIN {X 0,Y 130.107,Z 264.523,A -85,B 0,C 180,E1 -28090.062,E2 -28090.062} C_VEL
LIN {X 0,Y 132.023,Z 268.563,A -85,B 0,C 180,E1 -28094.844,E2 -28094.844} C_VEL
LIN {X 0,Y 133.957,Z 272.449,A -85,B 0,C 180,E1 -28098.348,E2 -28098.348} C_VEL
LIN {X 0,Y 136.598,Z 278.318,A -85,B 0,C 180,E1 -28102.243,E2 -28102.243} C_VEL
LIN {X 0,Y 138.002,Z 282.51,A -85,B 0,C 180,E1 -28104.152,E2 -28104.152} C_VEL
LIN {X 0,Y 135.904,Z 300.994,A -85,B 0,C 180,E1 -28104.855,E2 -28104.855} C_VEL
LIN {X 0,Y 133.195,Z 313.705,A -85,B 0,C 180,E1 -28105.558,E2 -28105.558} C_VEL
LIN {X 0,Y 129.628,Z 325.388,A -85,B 0,C 180,E1 -28106.546,E2 -28106.546} C_VEL
LIN {X 0,Y 124.418,Z 338.014,A -85,B 0,C 180,E1 -28108.041,E2 -28108.041} C_VEL
LIN {X 0,Y 118.645,Z 349.252,A -85,B 0,C 180,E1 -28109.966,E2 -28109.966} C_VEL
LIN {X 0,Y 112.323,Z 359.368,A -85,B 0,C 180,E1 -28112.361,E2 -28112.361} C_VEL
LIN {X 0,Y 105.562,Z 368.487,A -85,B 0,C 180,E1 -28115.356,E2 -28115.356} C_VEL
LIN {X 0,Y 97.9,Z 377.376,A -85,B 0,C 180,E1 -28119.49,E2 -28119.49} C_VEL
LIN {X 0,Y 91.762,Z 383.759,A -85,B 0,C 180,E1 -28123.802,E2 -28123.802} C_VEL
LIN {X 0,Y 85.609,Z 389.35,A -85,B 0,C 180,E1 -28128.946,E2 -28128.946} C_VEL
LIN {X 0,Y 80.004,Z 394.038,A -85,B 0,C 180,E1 -28135.179,E2 -28135.179} C_VEL
LIN {X 0,Y 75.413,Z 397.616,A -85,B 0,C 180,E1 -28142.225,E2 -28142.225} C_VEL
LIN {X 0,Y 73.115,Z 399.461,A -85,B 0,C 180,E1 -28147.386,E2 -28147.386} C_VEL
LIN {X 0,Y 71.4,Z 400.844,A -85,B 0,C 180,E1 -28152.823,E2 -28152.823} C_VEL
LIN {X 0,Y 69.658,Z 402.433,A -85,B 0,C 180,E1 -28164.207,E2 -28164.207} C_VEL
LIN {X 0,Y 69.581,Z 402.64,A -85,B 0,C 180,E1 -28169.997,E2 -28169.997} C_VEL
LIN {X 0,Y 69.657,Z 402.414,A -85,B 0,C 180,E1 -28175.788,E2 -28175.788} C_VEL
LIN {X 0,Y 71.404,Z 400.8,A -85,B 0,C 180,E1 -28187.171,E2 -28187.171} C_VEL
LIN {X 0,Y 73.126,Z 399.398,A -85,B 0,C 180,E1 -28192.605,E2 -28192.605} C_VEL
LIN {X 0,Y 76.826,Z 396.461,A -85,B 0,C 180,E1 -28200.204,E2 -28200.204} C_VEL
LIN {X 0,Y 81.793,Z 392.49,A -85,B 0,C 180,E1 -28206.972,E2 -28206.972} C_VEL
LIN {X 0,Y 88.803,Z 386.382,A -85,B 0,C 180,E1 -28213.823,E2 -28213.823} C_VEL
LIN {X 0,Y 95.499,Z 379.71,A -85,B 0,C 180,E1 -28218.961,E2 -28218.961} C_VEL
LIN {X 0,Y 102.905,Z 371.434,A -85,B 0,C 180,E1 -28223.363,E2 -28223.363} C_VEL
LIN {X 0,Y 109.548,Z 362.939,A -85,B 0,C 180,E1 -28226.508,E2 -28226.508} C_VEL
LIN {X 0,Y 116.497,Z 352.442,A -85,B 0,C 180,E1 -28229.275,E2 -28229.275} C_VEL
LIN {X 0,Y 122.252,Z 342.051,A -85,B 0,C 180,E1 -28231.24,E2 -28231.24} C_VEL
LIN {X 0,Y 127.365,Z 330.64,A -85,B 0,C 180,E1 -28232.84,E2 -28232.84} C_VEL
LIN {X 0,Y 131.445,Z 318.859,A -85,B 0,C 180,E1 -28234.01,E2 -28234.01} C_VEL
LIN {X 0,Y 134.786,Z 305.5,A -85,B 0,C 180,E1 -28234.889,E2 -28234.889} C_VEL
LIN {X 0,Y 136.678,Z 293.263,A -85,B 0,C 180,E1 -28235.407,E2 -28235.407} C_VEL
LIN {X 0,Y 137.747,Z 282.29,A -85,B 0,C 180,E1 -28235.8,E2 -28235.8} C_VEL
LIN {X 0,Y 136.419,Z 278.24,A -85,B 0,C 180,E1 -28237.607,E2 -28237.607} C_VEL
LIN {X 0,Y 133.779,Z 272.437,A -85,B 0,C 180,E1 -28241.453,E2 -28241.453} C_VEL
LIN {X 0,Y 131.488,Z 267.616,A -85,B 0,C 180,E1 -28245.688,E2 -28245.688} C_VEL
LIN {X 0,Y 129.583,Z 263.821,A -85,B 0,C 180,E1 -28250.636,E2 -28250.636} C_VEL
LIN {X 0,Y 128.617,Z 261.976,A -85,B 0,C 180,E1 -28254.709,E2 -28254.709} C_VEL
LIN {X 0,Y 128.312,Z 261.959,A -85,B 0,C 180,E1 -28256.442,E2 -28256.442} C_VEL
LIN {X 0,Y 127.896,Z 263.544,A -85,B 0,C 180,E1 -28258.694,E2 -28258.694} C_VEL
LIN {X 0,Y 127.482,Z 267.613,A -85,B 0,C 180,E1 -28262.607,E2 -28262.607} C_VEL
LIN {X 0,Y 127.531,Z 268.383,A -85,B 0,C 180,E1 -28263.794,E2 -28263.794} C_VEL
LIN {X 0,Y 128.825,Z 271.447,A -85,B 0,C 180,E1 -28270.037,E2 -28270.037} C_VEL
LIN {X 0,Y 130.402,Z 275.035,A -85,B 0,C 180,E1 -28274.235,E2 -28274.235} C_VEL
LIN {X 0,Y 131.983,Z 278.533,A -85,B 0,C 180,E1 -28277.379,E2 -28277.379} C_VEL
LIN {X 0,Y 134.275,Z 284.117,A -85,B 0,C 180,E1 -28281.116,E2 -28281.116} C_VEL
LIN {X 0,Y 134.685,Z 285.234,A -85,B 0,C 180,E1 -28281.724,E2 -28281.724} C_VEL
LIN {X 0,Y 132.764,Z 300.656,A -85,B 0,C 180,E1 -28282.291,E2 -28282.291} C_VEL
LIN {X 0,Y 129.78,Z 313.838,A -85,B 0,C 180,E1 -28282.992,E2 -28282.992} C_VEL
LIN {X 0,Y 125.987,Z 325.714,A -85,B 0,C 180,E1 -28284.075,E2 -28284.075} C_VEL
LIN {X 0,Y 120.718,Z 337.971,A -85,B 0,C 180,E1 -28285.533,E2 -28285.533} C_VEL
LIN {X 0,Y 114.79,Z 349.001,A -85,B 0,C 180,E1 -28287.413,E2 -28287.413} C_VEL
LIN {X 0,Y 108.959,Z 357.94,A -85,B 0,C 180,E1 -28289.458,E2 -28289.458} C_VEL
LIN {X 0,Y 101.914,Z 367.113,A -85,B 0,C 180,E1 -28292.359,E2 -28292.359} C_VEL
LIN {X 0,Y 94.186,Z 375.816,A -85,B 0,C 180,E1 -28296.383,E2 -28296.383} C_VEL
LIN {X 0,Y 86.54,Z 383.211,A -85,B 0,C 180,E1 -28301.31,E2 -28301.31} C_VEL
LIN {X 0,Y 80.822,Z 388.052,A -85,B 0,C 180,E1 -28305.925,E2 -28305.925} C_VEL
LIN {X 0,Y 74.642,Z 392.757,A -85,B 0,C 180,E1 -28312.269,E2 -28312.269} C_VEL
LIN {X 0,Y 69.642,Z 396.355,A -85,B 0,C 180,E1 -28319.7,E2 -28319.7} C_VEL
LIN {X 0,Y 66.976,Z 398.213,A -85,B 0,C 180,E1 -28325.186,E2 -28325.186} C_VEL
LIN {X 0,Y 64.898,Z 399.607,A -85,B 0,C 180,E1 -28331.045,E2 -28331.045} C_VEL
LIN {X 0,Y 62.688,Z 401.207,A -85,B 0,C 180,E1 -28343.566,E2 -28343.566} C_VEL
LIN {X 0,Y 62.554,Z 401.431,A -85,B 0,C 180,E1 -28350.003,E2 -28350.003} C_VEL
LIN {X 0,Y 62.688,Z 401.233,A -85,B 0,C 180,E1 -28356.44,E2 -28356.44} C_VEL
LIN {X 0,Y 64.899,Z 399.667,A -85,B 0,C 180,E1 -28368.96,E2 -28368.96} C_VEL
LIN {X 0,Y 66.973,Z 398.299,A -85,B 0,C 180,E1 -28374.821,E2 -28374.821} C_VEL
LIN {X 0,Y 71.109,Z 395.412,A -85,B 0,C 180,E1 -28382.93,E2 -28382.93} C_VEL
LIN {X 0,Y 76.547,Z 391.497,A -85,B 0,C 180,E1 -28389.995,E2 -28389.995} C_VEL
LIN {X 0,Y 82.985,Z 386.448,A -85,B 0,C 180,E1 -28396.045,E2 -28396.045} C_VEL
LIN {X 0,Y 90.152,Z 380.09,A -85,B 0,C 180,E1 -28401.223,E2 -28401.223} C_VEL
LIN {X 0,Y 97.766,Z 372.143,A -85,B 0,C 180,E1 -28405.761,E2 -28405.761} C_VEL
LIN {X 0,Y 104.642,Z 364.04,A -85,B 0,C 180,E1 -28408.907,E2 -28408.907} C_VEL
LIN {X 0,Y 111.798,Z 354.153,A -85,B 0,C 180,E1 -28411.653,E2 -28411.653} C_VEL
LIN {X 0,Y 118.444,Z 343.013,A -85,B 0,C 180,E1 -28413.826,E2 -28413.826} C_VEL
LIN {X 0,Y 123.68,Z 332.095,A -85,B 0,C 180,E1 -28415.394,E2 -28415.394} C_VEL
LIN {X 0,Y 128.256,Z 320.02,A -85,B 0,C 180,E1 -28416.613,E2 -28416.613} C_VEL
LIN {X 0,Y 131.767,Z 307.113,A -85,B 0,C 180,E1 -28417.543,E2 -28417.543} C_VEL
LIN {X 0,Y 133.954,Z 294.459,A -85,B 0,C 180,E1 -28418.128,E2 -28418.128} C_VEL
LIN {X 0,Y 134.901,Z 285.288,A -85,B 0,C 180,E1 -28418.487,E2 -28418.487} C_VEL
LIN {X 0,Y 132.539,Z 279.37,A -85,B 0,C 180,E1 -28422.26,E2 -28422.26} C_VEL
LIN {X 0,Y 131.006,Z 276.03,A -85,B 0,C 180,E1 -28425.187,E2 -28425.187} C_VEL
LIN {X 0,Y 129.782,Z 273.348,A -85,B 0,C 180,E1 -28428.085,E2 -28428.085} C_VEL
LIN {X 0,Y 128.817,Z 270.905,A -85,B 0,C 180,E1 -28431.173,E2 -28431.173} C_VEL
LIN {X 0,Y 127.759,Z 267.209,A -85,B 0,C 180,E1 -28440,E2 -28440} C_VEL
LIN {X 0,Y 128.991,Z 271.435,A -85,B 0,C 180,E1 -28449.407,E2 -28449.407} C_VEL
LIN {X 0,Y 130.676,Z 275.283,A -85,B 0,C 180,E1 -28454.006,E2 -28454.006} C_VEL
LIN {X 0,Y 132.656,Z 279.631,A -85,B 0,C 180,E1 -28457.86,E2 -28457.86} C_VEL
LIN {X 0,Y 134.867,Z 285.298,A -85,B 0,C 180,E1 -28461.394,E2 -28461.394} C_VEL
LIN {X 0,Y 134.936,Z 286.083,A -85,B 0,C 180,E1 -28461.58,E2 -28461.58} C_VEL
LIN {X 0,Y 132.803,Z 302.508,A -85,B 0,C 180,E1 -28462.136,E2 -28462.136} C_VEL
LIN {X 0,Y 130.063,Z 314.543,A -85,B 0,C 180,E1 -28462.805,E2 -28462.805} C_VEL
LIN {X 0,Y 125.846,Z 327.323,A -85,B 0,C 180,E1 -28463.868,E2 -28463.868} C_VEL
LIN {X 0,Y 120.489,Z 339.536,A -85,B 0,C 180,E1 -28465.298,E2 -28465.298} C_VEL
LIN {X 0,Y 114.534,Z 350.431,A -85,B 0,C 180,E1 -28467.158,E2 -28467.158} C_VEL
LIN {X 0,Y 107.244,Z 361.258,A -85,B 0,C 180,E1 -28469.737,E2 -28469.737} C_VEL
LIN {X 0,Y 100.224,Z 370.053,A -85,B 0,C 180,E1 -28472.703,E2 -28472.703} C_VEL
LIN {X 0,Y 92.238,Z 378.621,A -85,B 0,C 180,E1 -28476.865,E2 -28476.865} C_VEL
LIN {X 0,Y 84.975,Z 385.478,A -85,B 0,C 180,E1 -28481.894,E2 -28481.894} C_VEL
LIN {X 0,Y 78.233,Z 390.968,A -85,B 0,C 180,E1 -28487.641,E2 -28487.641} C_VEL
LIN {X 0,Y 72.46,Z 395.273,A -85,B 0,C 180,E1 -28494.41,E2 -28494.41} C_VEL
LIN {X 0,Y 69.185,Z 397.552,A -85,B 0,C 180,E1 -28499.473,E2 -28499.473} C_VEL
LIN {X 0,Y 66.603,Z 399.396,A -85,B 0,C 180,E1 -28505.032,E2 -28505.032} C_VEL
LIN {X 0,Y 63.29,Z 401.767,A -85,B 0,C 180,E1 -28517.166,E2 -28517.166} C_VEL
LIN {X 0,Y 62.589,Z 402.368,A -85,B 0,C 180,E1 -28523.55,E2 -28523.55} C_VEL
LIN {X 0,Y 62.5,Z 402.575,A -85,B 0,C 180,E1 -28529.997,E2 -28529.997} C_VEL
LIN {X 0,Y 62.589,Z 402.348,A -85,B 0,C 180,E1 -28536.444,E2 -28536.444} C_VEL
LIN {X 0,Y 63.289,Z 401.735,A -85,B 0,C 180,E1 -28542.829,E2 -28542.829} C_VEL
LIN {X 0,Y 64.625,Z 400.735,A -85,B 0,C 180,E1 -28549.038,E2 -28549.038} C_VEL
LIN {X 0,Y 66.611,Z 399.332,A -85,B 0,C 180,E1 -28554.959,E2 -28554.959} C_VEL
LIN {X 0,Y 70.751,Z 396.395,A -85,B 0,C 180,E1 -28563.112,E2 -28563.112} C_VEL
LIN {X 0,Y 76.217,Z 392.424,A -85,B 0,C 180,E1 -28570.197,E2 -28570.197} C_VEL
LIN {X 0,Y 83.813,Z 386.315,A -85,B 0,C 180,E1 -28577.194,E2 -28577.194} C_VEL
LIN {X 0,Y 90.973,Z 379.643,A -85,B 0,C 180,E1 -28582.353,E2 -28582.353} C_VEL
LIN {X 0,Y 98.825,Z 371.367,A -85,B 0,C 180,E1 -28586.674,E2 -28586.674} C_VEL
LIN {X 0,Y 105.792,Z 362.871,A -85,B 0,C 180,E1 -28589.72,E2 -28589.72} C_VEL
LIN {X 0,Y 113.027,Z 352.374,A -85,B 0,C 180,E1 -28592.377,E2 -28592.377} C_VEL
LIN {X 0,Y 118.994,Z 341.981,A -85,B 0,C 180,E1 -28594.243,E2 -28594.243} C_VEL
LIN {X 0,Y 124.291,Z 330.569,A -85,B 0,C 180,E1 -28595.746,E2 -28595.746} C_VEL
LIN {X 0,Y 128.682,Z 318.175,A -85,B 0,C 180,E1 -28596.893,E2 -28596.893} C_VEL
LIN {X 0,Y 132.123,Z 304.552,A -85,B 0,C 180,E1 -28597.717,E2 -28597.717} C_VEL
LIN {X 0,Y 134.064,Z 291.525,A -85,B 0,C 180,E1 -28598.225,E2 -28598.225} C_VEL
LIN {X 0,Y 134.671,Z 285.206,A -85,B 0,C 180,E1 -28598.468,E2 -28598.468} C_VEL
LIN {X 0,Y 132.37,Z 279.341,A -85,B 0,C 180,E1 -28602.125,E2 -28602.125} C_VEL
LIN {X 0,Y 130.072,Z 274.179,A -85,B 0,C 180,E1 -28606.728,E2 -28606.728} C_VEL
LIN {X 0,Y 128.475,Z 270.67,A -85,B 0,C 180,E1 -28611.348,E2 -28611.348} C_VEL
LIN {X 0,Y 127.454,Z 266.911,A -85,B 0,C 180,E1 -28619.408,E2 -28619.408} C_VEL
LIN {X 0,Y 127.448,Z 267.236,A -85,B 0,C 180,E1 -28621.58,E2 -28621.58} C_VEL
LIN {X 0,Y 127.531,Z 268.383,A -85,B 0,C 180,E1 -28623.794,E2 -28623.794} C_VEL
LIN {X 0,Y 127.782,Z 270.283,A -85,B 0,C 180,E1 -28626.304,E2 -28626.304} C_VEL
LIN {X 0,Y 128.098,Z 273.166,A -85,B 0,C 180,E1 -28628.63,E2 -28628.63} C_VEL
LIN {X 0,Y 129.068,Z 280.199,A -85,B 0,C 180,E1 -28632.982,E2 -28632.982} C_VEL
LIN {X 0,Y 130.226,Z 284.575,A -85,B 0,C 180,E1 -28635.936,E2 -28635.936} C_VEL
LIN {X 0,Y 131.833,Z 288.881,A -85,B 0,C 180,E1 -28638.958,E2 -28638.958} C_VEL
LIN {X 0,Y 129.964,Z 302.35,A -85,B 0,C 180,E1 -28639.474,E2 -28639.474} C_VEL
LIN {X 0,Y 126.66,Z 315.643,A -85,B 0,C 180,E1 -28640.178,E2 -28640.178} C_VEL
LIN {X 0,Y 122.409,Z 327.989,A -85,B 0,C 180,E1 -28641.292,E2 -28641.292} C_VEL
LIN {X 0,Y 117.071,Z 339.602,A -85,B 0,C 180,E1 -28642.64,E2 -28642.64} C_VEL
LIN {X 0,Y 110.94,Z 350.25,A -85,B 0,C 180,E1 -28644.412,E2 -28644.412} C_VEL
LIN {X 0,Y 104.154,Z 359.964,A -85,B 0,C 180,E1 -28646.618,E2 -28646.618} C_VEL
LIN {X 0,Y 96.866,Z 368.805,A -85,B 0,C 180,E1 -28649.472,E2 -28649.472} C_VEL
LIN {X 0,Y 88.616,Z 377.391,A -85,B 0,C 180,E1 -28653.567,E2 -28653.567} C_VEL
LIN {X 0,Y 80.74,Z 384.304,A -85,B 0,C 180,E1 -28658.432,E2 -28658.432} C_VEL
LIN {X 0,Y 73.537,Z 389.812,A -85,B 0,C 180,E1 -28664.215,E2 -28664.215} C_VEL
LIN {X 0,Y 67.121,Z 394.135,A -85,B 0,C 180,E1 -28671.084,E2 -28671.084} C_VEL
LIN {X 0,Y 63.579,Z 396.421,A -85,B 0,C 180,E1 -28676.452,E2 -28676.452} C_VEL
LIN {X 0,Y 60.581,Z 398.279,A -85,B 0,C 180,E1 -28682.356,E2 -28682.356} C_VEL
LIN {X 0,Y 58.219,Z 399.672,A -85,B 0,C 180,E1 -28688.771,E2 -28688.771} C_VEL
LIN {X 0,Y 56.58,Z 400.664,A -85,B 0,C 180,E1 -28695.619,E2 -28695.619} C_VEL
LIN {X 0,Y 55.474,Z 401.496,A -85,B 0,C 180,E1 -28710.003,E2 -28710.003} C_VEL
LIN {X 0,Y 55.632,Z 401.298,A -85,B 0,C 180,E1 -28717.261,E2 -28717.261} C_VEL
LIN {X 0,Y 56.581,Z 400.706,A -85,B 0,C 180,E1 -28724.387,E2 -28724.387} C_VEL
LIN {X 0,Y 60.576,Z 398.363,A -85,B 0,C 180,E1 -28737.653,E2 -28737.653} C_VEL
LIN {X 0,Y 65.241,Z 395.476,A -85,B 0,C 180,E1 -28746.336,E2 -28746.336} C_VEL
LIN {X 0,Y 71.246,Z 391.561,A -85,B 0,C 180,E1 -28753.673,E2 -28753.673} C_VEL
LIN {X 0,Y 78.206,Z 386.512,A -85,B 0,C 180,E1 -28759.807,E2 -28759.807} C_VEL
LIN {X 0,Y 86.372,Z 379.657,A -85,B 0,C 180,E1 -28765.279,E2 -28765.279} C_VEL
LIN {X 0,Y 93.945,Z 372.206,A -85,B 0,C 180,E1 -28769.353,E2 -28769.353} C_VEL
LIN {X 0,Y 101.158,Z 364.102,A -85,B 0,C 180,E1 -28772.353,E2 -28772.353} C_VEL
LIN {X 0,Y 108.614,Z 354.215,A -85,B 0,C 180,E1 -28774.943,E2 -28774.943} C_VEL
LIN {X 0,Y 115.493,Z 343.073,A -85,B 0,C 180,E1 -28776.983,E2 -28776.983} C_VEL
LIN {X 0,Y 120.895,Z 332.155,A -85,B 0,C 180,E1 -28778.456,E2 -28778.456} C_VEL
LIN {X 0,Y 125.438,Z 320.55,A -85,B 0,C 180,E1 -28779.554,E2 -28779.554} C_VEL
LIN {X 0,Y 129.135,Z 307.57,A -85,B 0,C 180,E1 -28780.433,E2 -28780.433} C_VEL
LIN {X 0,Y 131.428,Z 294.894,A -85,B 0,C 180,E1 -28780.983,E2 -28780.983} C_VEL
LIN {X 0,Y 132.103,Z 289.111,A -85,B 0,C 180,E1 -28781.178,E2 -28781.178} C_VEL
LIN {X 0,Y 130.118,Z 283.748,A -85,B 0,C 180,E1 -28785.034,E2 -28785.034} C_VEL
LIN {X 0,Y 128.477,Z 279.889,A -85,B 0,C 180,E1 -28789.161,E2 -28789.161} C_VEL
LIN {X 0,Y 127.673,Z 277.7,A -85,B 0,C 180,E1 -28792.091,E2 -28792.091} C_VEL
LIN {X 0,Y 126.878,Z 274.389,A -85,B 0,C 180,E1 -28800,E2 -28800} C_VEL
LIN {X 0,Y 127.832,Z 278.149,A -85,B 0,C 180,E1 -28808.496,E2 -28808.496} C_VEL
LIN {X 0,Y 129.239,Z 281.744,A -85,B 0,C 180,E1 -28812.863,E2 -28812.863} C_VEL
LIN {X 0,Y 130.913,Z 285.791,A -85,B 0,C 180,E1 -28816.526,E2 -28816.526} C_VEL
LIN {X 0,Y 132.108,Z 289.123,A -85,B 0,C 180,E1 -28818.747,E2 -28818.747} C_VEL
LIN {X 0,Y 130.216,Z 302.962,A -85,B 0,C 180,E1 -28819.274,E2 -28819.274} C_VEL
LIN {X 0,Y 127.1,Z 315.741,A -85,B 0,C 180,E1 -28819.946,E2 -28819.946} C_VEL
LIN {X 0,Y 123.088,Z 327.424,A -85,B 0,C 180,E1 -28820.869,E2 -28820.869} C_VEL
LIN {X 0,Y 117.638,Z 339.477,A -85,B 0,C 180,E1 -28822.178,E2 -28822.178} C_VEL
LIN {X 0,Y 111.472,Z 350.37,A -85,B 0,C 180,E1 -28823.909,E2 -28823.909} C_VEL
LIN {X 0,Y 103.905,Z 361.196,A -85,B 0,C 180,E1 -28826.335,E2 -28826.335} C_VEL
LIN {X 0,Y 96.571,Z 369.991,A -85,B 0,C 180,E1 -28829.154,E2 -28829.154} C_VEL
LIN {X 0,Y 89.524,Z 377.25,A -85,B 0,C 180,E1 -28832.442,E2 -28832.442} C_VEL
LIN {X 0,Y 82.741,Z 383.442,A -85,B 0,C 180,E1 -28836.483,E2 -28836.483} C_VEL
LIN {X 0,Y 75.468,Z 389.223,A -85,B 0,C 180,E1 -28841.839,E2 -28841.839} C_VEL
LIN {X 0,Y 68.8,Z 393.91,A -85,B 0,C 180,E1 -28848.393,E2 -28848.393} C_VEL
LIN {X 0,Y 63.148,Z 397.488,A -85,B 0,C 180,E1 -28856.185,E2 -28856.185} C_VEL
LIN {X 0,Y 60.215,Z 399.332,A -85,B 0,C 180,E1 -28862.167,E2 -28862.167} C_VEL
LIN {X 0,Y 56.369,Z 401.702,A -85,B 0,C 180,E1 -28875.558,E2 -28875.558} C_VEL
LIN {X 0,Y 55.546,Z 402.303,A -85,B 0,C 180,E1 -28882.728,E2 -28882.728} C_VEL
LIN {X 0,Y 55.402,Z 402.511,A -85,B 0,C 180,E1 -28889.997,E2 -28889.997} C_VEL
LIN {X 0,Y 55.545,Z 402.283,A -85,B 0,C 180,E1 -28897.266,E2 -28897.266} C_VEL
LIN {X 0,Y 57.94,Z 400.669,A -85,B 0,C 180,E1 -28911.336,E2 -28911.336} C_VEL
LIN {X 0,Y 60.221,Z 399.266,A -85,B 0,C 180,E1 -28917.824,E2 -28917.824} C_VEL
LIN {X 0,Y 64.901,Z 396.329,A -85,B 0,C 180,E1 -28926.55,E2 -28926.55} C_VEL
LIN {X 0,Y 70.91,Z 392.357,A -85,B 0,C 180,E1 -28933.925,E2 -28933.925} C_VEL
LIN {X 0,Y 79.135,Z 386.248,A -85,B 0,C 180,E1 -28940.99,E2 -28940.99} C_VEL
LIN {X 0,Y 86.797,Z 379.576,A -85,B 0,C 180,E1 -28946.087,E2 -28946.087} C_VEL
LIN {X 0,Y 95.104,Z 371.299,A -85,B 0,C 180,E1 -28950.255,E2 -28950.255} C_VEL
LIN {X 0,Y 102.393,Z 362.803,A -85,B 0,C 180,E1 -28953.156,E2 -28953.156} C_VEL
LIN {X 0,Y 109.907,Z 352.305,A -85,B 0,C 180,E1 -28955.667,E2 -28955.667} C_VEL
LIN {X 0,Y 116.862,Z 340.481,A -85,B 0,C 180,E1 -28957.607,E2 -28957.607} C_VEL
LIN {X 0,Y 122.228,Z 328.809,A -85,B 0,C 180,E1 -28958.964,E2 -28958.964} C_VEL
LIN {X 0,Y 126.658,Z 316.191,A -85,B 0,C 180,E1 -28959.979,E2 -28959.979} C_VEL
LIN {X 0,Y 129.727,Z 303.89,A -85,B 0,C 180,E1 -28960.647,E2 -28960.647} C_VEL
LIN {X 0,Y 131.733,Z 290.154,A -85,B 0,C 180,E1 -28961.133,E2 -28961.133} C_VEL
LIN {X 0,Y 131.766,Z 288.676,A -85,B 0,C 180,E1 -28961.336,E2 -28961.336} C_VEL
LIN {X 0,Y 129.864,Z 283.626,A -85,B 0,C 180,E1 -28965.007,E2 -28965.007} C_VEL
LIN {X 0,Y 128.274,Z 279.853,A -85,B 0,C 180,E1 -28968.944,E2 -28968.944} C_VEL
LIN {X 0,Y 127.336,Z 277.434,A -85,B 0,C 180,E1 -28972.269,E2 -28972.269} C_VEL
LIN {X 0,Y 126.59,Z 273.877,A -85,B 0,C 180,E1 -28980,E2 -28980} C_VEL
LIN {X 0,Y 127.632,Z 278.1,A -85,B 0,C 180,E1 -28989.059,E2 -28989.059} C_VEL
LIN {X 0,Y 129.074,Z 281.768,A -85,B 0,C 180,E1 -28993.37,E2 -28993.37} C_VEL
LIN {X 0,Y 130.226,Z 284.575,A -85,B 0,C 180,E1 -28995.936,E2 -28995.936} C_VEL
LIN {X 0,Y 130.526,Z 286.276,A -85,B 0,C 180,E1 -28996.708,E2 -28996.708} C_VEL
LIN {X 0,Y 130.529,Z 289.201,A -85,B 0,C 180,E1 -28997.249,E2 -28997.249} C_VEL
LIN {X 0,Y 130.195,Z 292.464,A -85,B 0,C 180,E1 -28997.409,E2 -28997.409} C_VEL
LIN {X 0,Y 129.352,Z 296.747,A -85,B 0,C 180,E1 -28997.142,E2 -28997.142} C_VEL
LIN {X 0,Y 127.44,Z 304.099,A -85,B 0,C 180,E1 -28996.572,E2 -28996.572} C_VEL
LIN {X 0,Y 127.079,Z 305.589,A -85,B 0,C 180,E1 -28996.598,E2 -28996.598} C_VEL
LIN {X 0,Y 123.513,Z 318.569,A -85,B 0,C 180,E1 -28997.306,E2 -28997.306} C_VEL
LIN {X 0,Y 119.221,Z 329.958,A -85,B 0,C 180,E1 -28998.304,E2 -28998.304} C_VEL
LIN {X 0,Y 113.729,Z 341.103,A -85,B 0,C 180,E1 -28999.552,E2 -28999.552} C_VEL
LIN {X 0,Y 106.622,Z 352.664,A -85,B 0,C 180,E1 -29001.409,E2 -29001.409} C_VEL
LIN {X 0,Y 99.651,Z 361.979,A -85,B 0,C 180,E1 -29003.539,E2 -29003.539} C_VEL
LIN {X 0,Y 92.083,Z 370.466,A -85,B 0,C 180,E1 -29006.268,E2 -29006.268} C_VEL
LIN {X 0,Y 83.008,Z 379.096,A -85,B 0,C 180,E1 -29010.531,E2 -29010.531} C_VEL
LIN {X 0,Y 75.174,Z 385.376,A -85,B 0,C 180,E1 -29015.117,E2 -29015.117} C_VEL
LIN {X 0,Y 66.324,Z 391.468,A -85,B 0,C 180,E1 -29022.125,E2 -29022.125} C_VEL
LIN {X 0,Y 59.682,Z 395.424,A -85,B 0,C 180,E1 -29029.639,E2 -29029.639} C_VEL
LIN {X 0,Y 54.37,Z 398.344,A -85,B 0,C 180,E1 -29038.87,E2 -29038.87} C_VEL
LIN {X 0,Y 51.662,Z 399.738,A -85,B 0,C 180,E1 -29045.918,E2 -29045.918} C_VEL
LIN {X 0,Y 49.726,Z 400.729,A -85,B 0,C 180,E1 -29053.585,E2 -29053.585} C_VEL
LIN {X 0,Y 48.376,Z 401.561,A -85,B 0,C 180,E1 -29070.004,E2 -29070.004} C_VEL
LIN {X 0,Y 48.605,Z 401.362,A -85,B 0,C 180,E1 -29078.317,E2 -29078.317} C_VEL
LIN {X 0,Y 49.728,Z 400.771,A -85,B 0,C 180,E1 -29086.422,E2 -29086.422} C_VEL
LIN {X 0,Y 54.364,Z 398.428,A -85,B 0,C 180,E1 -29101.142,E2 -29101.142} C_VEL
LIN {X 0,Y 59.655,Z 395.541,A -85,B 0,C 180,E1 -29110.39,E2 -29110.39} C_VEL
LIN {X 0,Y 66.288,Z 391.625,A -85,B 0,C 180,E1 -29117.918,E2 -29117.918} C_VEL
LIN {X 0,Y 73.813,Z 386.576,A -85,B 0,C 180,E1 -29124.031,E2 -29124.031} C_VEL
LIN {X 0,Y 81.961,Z 380.217,A -85,B 0,C 180,E1 -29129.036,E2 -29129.036} C_VEL
LIN {X 0,Y 90.52,Z 372.269,A -85,B 0,C 180,E1 -29133.236,E2 -29133.236} C_VEL
LIN {X 0,Y 98.06,Z 364.164,A -85,B 0,C 180,E1 -29136.037,E2 -29136.037} C_VEL
LIN {X 0,Y 105.803,Z 354.276,A -85,B 0,C 180,E1 -29138.428,E2 -29138.428} C_VEL
LIN {X 0,Y 112.907,Z 343.134,A -85,B 0,C 180,E1 -29140.301,E2 -29140.301} C_VEL
LIN {X 0,Y 118.478,Z 332.214,A -85,B 0,C 180,E1 -29141.642,E2 -29141.642} C_VEL
LIN {X 0,Y 123.31,Z 320.133,A -85,B 0,C 180,E1 -29142.682,E2 -29142.682} C_VEL
LIN {X 0,Y 126.937,Z 307.623,A -85,B 0,C 180,E1 -29143.449,E2 -29143.449} C_VEL
LIN {X 0,Y 129.369,Z 294.297,A -85,B 0,C 180,E1 -29143.985,E2 -29143.985} C_VEL
LIN {X 0,Y 129.49,Z 292.786,A -85,B 0,C 180,E1 -29144.153,E2 -29144.153} C_VEL
LIN {X 0,Y 128.173,Z 289.094,A -85,B 0,C 180,E1 -29147.33,E2 -29147.33} C_VEL
LIN {X 0,Y 127.273,Z 286.592,A -85,B 0,C 180,E1 -29150.063,E2 -29150.063} C_VEL
LIN {X 0,Y 126.515,Z 284.373,A -85,B 0,C 180,E1 -29153.261,E2 -29153.261} C_VEL
LIN {X 0,Y 125.998,Z 281.556,A -85,B 0,C 180,E1 -29160,E2 -29160} C_VEL
LIN {X 0,Y 126.756,Z 285.062,A -85,B 0,C 180,E1 -29167.813,E2 -29167.813} C_VEL
LIN {X 0,Y 127.919,Z 288.417,A -85,B 0,C 180,E1 -29171.89,E2 -29171.89} C_VEL
LIN {X 0,Y 129.329,Z 292.261,A -85,B 0,C 180,E1 -29175.362,E2 -29175.362} C_VEL
LIN {X 0,Y 129.568,Z 293.053,A -85,B 0,C 180,E1 -29175.922,E2 -29175.922} C_VEL
LIN {X 0,Y 127.416,Z 305.835,A -85,B 0,C 180,E1 -29176.394,E2 -29176.394} C_VEL
LIN {X 0,Y 123.77,Z 319.18,A -85,B 0,C 180,E1 -29177.104,E2 -29177.104} C_VEL
LIN {X 0,Y 119.099,Z 331.238,A -85,B 0,C 180,E1 -29178.042,E2 -29178.042} C_VEL
LIN {X 0,Y 112.737,Z 343.777,A -85,B 0,C 180,E1 -29179.457,E2 -29179.457} C_VEL
LIN {X 0,Y 105.627,Z 354.947,A -85,B 0,C 180,E1 -29181.329,E2 -29181.329} C_VEL
LIN {X 0,Y 97.869,Z 364.857,A -85,B 0,C 180,E1 -29183.711,E2 -29183.711} C_VEL
LIN {X 0,Y 88.837,Z 374.465,A -85,B 0,C 180,E1 -29187.125,E2 -29187.125} C_VEL
LIN {X 0,Y 80.331,Z 382.039,A -85,B 0,C 180,E1 -29191.31,E2 -29191.31} C_VEL
LIN {X 0,Y 73.541,Z 387.347,A -85,B 0,C 180,E1 -29195.675,E2 -29195.675} C_VEL
LIN {X 0,Y 65.964,Z 392.419,A -85,B 0,C 180,E1 -29201.769,E2 -29201.769} C_VEL
LIN {X 0,Y 59.339,Z 396.357,A -85,B 0,C 180,E1 -29209.349,E2 -29209.349} C_VEL
LIN {X 0,Y 54.019,Z 399.267,A -85,B 0,C 180,E1 -29218.638,E2 -29218.638} C_VEL
LIN {X 0,Y 49.516,Z 401.637,A -85,B 0,C 180,E1 -29233.505,E2 -29233.505} C_VEL
LIN {X 0,Y 48.505,Z 402.239,A -85,B 0,C 180,E1 -29241.666,E2 -29241.666} C_VEL
LIN {X 0,Y 48.319,Z 402.446,A -85,B 0,C 180,E1 -29249.996,E2 -29249.996} C_VEL
LIN {X 0,Y 48.505,Z 402.218,A -85,B 0,C 180,E1 -29258.327,E2 -29258.327} C_VEL
LIN {X 0,Y 51.38,Z 400.604,A -85,B 0,C 180,E1 -29274.223,E2 -29274.223} C_VEL
LIN {X 0,Y 54.023,Z 399.201,A -85,B 0,C 180,E1 -29281.353,E2 -29281.353} C_VEL
LIN {X 0,Y 59.333,Z 396.263,A -85,B 0,C 180,E1 -29290.648,E2 -29290.648} C_VEL
LIN {X 0,Y 65.953,Z 392.291,A -85,B 0,C 180,E1 -29298.233,E2 -29298.233} C_VEL
LIN {X 0,Y 74.853,Z 386.181,A -85,B 0,C 180,E1 -29305.233,E2 -29305.233} C_VEL
LIN {X 0,Y 83.027,Z 379.508,A -85,B 0,C 180,E1 -29310.178,E2 -29310.178} C_VEL
LIN {X 0,Y 91.791,Z 371.232,A -85,B 0,C 180,E1 -29314.104,E2 -29314.104} C_VEL
LIN {X 0,Y 99.389,Z 362.735,A -85,B 0,C 180,E1 -29316.81,E2 -29316.81} C_VEL
LIN {X 0,Y 107.174,Z 352.236,A -85,B 0,C 180,E1 -29319.131,E2 -29319.131} C_VEL
LIN {X 0,Y 114.35,Z 340.411,A -85,B 0,C 180,E1 -29320.892,E2 -29320.892} C_VEL
LIN {X 0,Y 119.757,Z 329.012,A -85,B 0,C 180,E1 -29322.101,E2 -29322.101} C_VEL
LIN {X 0,Y 124.385,Z 316.199,A -85,B 0,C 180,E1 -29323.042,E2 -29323.042} C_VEL
LIN {X 0,Y 127.583,Z 303.689,A -85,B 0,C 180,E1 -29323.654,E2 -29323.654} C_VEL
LIN {X 0,Y 129.264,Z 292.732,A -85,B 0,C 180,E1 -29324.102,E2 -29324.102} C_VEL
LIN {X 0,Y 127.914,Z 288.91,A -85,B 0,C 180,E1 -29327.304,E2 -29327.304} C_VEL
LIN {X 0,Y 126.882,Z 286.123,A -85,B 0,C 180,E1 -29330.435,E2 -29330.435} C_VEL
LIN {X 0,Y 126.232,Z 284.19,A -85,B 0,C 180,E1 -29333.206,E2 -29333.206} C_VEL
LIN {X 0,Y 125.715,Z 280.996,A -85,B 0,C 180,E1 -29340,E2 -29340} C_VEL
LIN {X 0,Y 126.545,Z 285.02,A -85,B 0,C 180,E1 -29348.383,E2 -29348.383} C_VEL
LIN {X 0,Y 127.712,Z 288.324,A -85,B 0,C 180,E1 -29352.313,E2 -29352.313} C_VEL
LIN {X 0,Y 129.093,Z 292.177,A -85,B 0,C 180,E1 -29355.695,E2 -29355.695} C_VEL
LIN {X 0,Y 129.277,Z 292.794,A -85,B 0,C 180,E1 -29356.129,E2 -29356.129} C_VEL
LIN {X 0,Y 127.079,Z 305.589,A -85,B 0,C 180,E1 -29356.598,E2 -29356.598} C_VEL
LIN {X 0,Y 125.485,Z 311.284,A -85,B 0,C 180,E1 -29356.551,E2 -29356.551} C_VEL
LIN {X 0,Y 121.878,Z 320.4,A -85,B 0,C 180,E1 -29355.847,E2 -29355.847} C_VEL
LIN {X 0,Y 117.667,Z 329.316,A -85,B 0,C 180,E1 -29355.247,E2 -29355.247} C_VEL
LIN {X 0,Y 115.043,Z 334.568,A -85,B 0,C 180,E1 -29355.395,E2 -29355.395} C_VEL
LIN {X 0,Y 109.096,Z 345.353,A -85,B 0,C 180,E1 -29356.625,E2 -29356.625} C_VEL
LIN {X 0,Y 101.817,Z 356.022,A -85,B 0,C 180,E1 -29358.368,E2 -29358.368} C_VEL
LIN {X 0,Y 93.854,Z 365.63,A -85,B 0,C 180,E1 -29360.613,E2 -29360.613} C_VEL
LIN {X 0,Y 86.093,Z 373.499,A -85,B 0,C 180,E1 -29363.319,E2 -29363.319} C_VEL
LIN {X 0,Y 77.434,Z 380.964,A -85,B 0,C 180,E1 -29367.207,E2 -29367.207} C_VEL
LIN {X 0,Y 69.908,Z 386.44,A -85,B 0,C 180,E1 -29371.3,E2 -29371.3} C_VEL
LIN {X 0,Y 61.785,Z 391.534,A -85,B 0,C 180,E1 -29377.233,E2 -29377.233} C_VEL
LIN {X 0,Y 54.458,Z 395.49,A -85,B 0,C 180,E1 -29384.788,E2 -29384.788} C_VEL
LIN {X 0,Y 48.418,Z 398.41,A -85,B 0,C 180,E1 -29394.511,E2 -29394.511} C_VEL
LIN {X 0,Y 45.276,Z 399.803,A -85,B 0,C 180,E1 -29402.251,E2 -29402.251} C_VEL
LIN {X 0,Y 42.966,Z 400.794,A -85,B 0,C 180,E1 -29410.909,E2 -29410.909} C_VEL
LIN {X 0,Y 41.294,Z 401.626,A -85,B 0,C 180,E1 -29430.004,E2 -29430.004} C_VEL
LIN {X 0,Y 41.589,Z 401.427,A -85,B 0,C 180,E1 -29439.733,E2 -29439.733} C_VEL
LIN {X 0,Y 42.967,Z 400.835,A -85,B 0,C 180,E1 -29449.099,E2 -29449.099} C_VEL
LIN {X 0,Y 48.41,Z 398.492,A -85,B 0,C 180,E1 -29465.504,E2 -29465.504} C_VEL
LIN {X 0,Y 54.435,Z 395.605,A -85,B 0,C 180,E1 -29475.246,E2 -29475.246} C_VEL
LIN {X 0,Y 61.754,Z 391.688,A -85,B 0,C 180,E1 -29482.814,E2 -29482.814} C_VEL
LIN {X 0,Y 69.875,Z 386.639,A -85,B 0,C 180,E1 -29488.754,E2 -29488.754} C_VEL
LIN {X 0,Y 78.538,Z 380.28,A -85,B 0,C 180,E1 -29493.492,E2 -29493.492} C_VEL
LIN {X 0,Y 87.549,Z 372.332,A -85,B 0,C 180,E1 -29497.394,E2 -29497.394} C_VEL
LIN {X 0,Y 95.392,Z 364.227,A -85,B 0,C 180,E1 -29499.945,E2 -29499.945} C_VEL
LIN {X 0,Y 103.402,Z 354.338,A -85,B 0,C 180,E1 -29502.092,E2 -29502.092} C_VEL
LIN {X 0,Y 110.718,Z 343.194,A -85,B 0,C 180,E1 -29503.757,E2 -29503.757} C_VEL
LIN {X 0,Y 116.442,Z 332.273,A -85,B 0,C 180,E1 -29504.95,E2 -29504.95} C_VEL
LIN {X 0,Y 121.386,Z 320.203,A -85,B 0,C 180,E1 -29505.874,E2 -29505.874} C_VEL
LIN {X 0,Y 125.158,Z 307.408,A -85,B 0,C 180,E1 -29506.583,E2 -29506.583} C_VEL
LIN {X 0,Y 127.214,Z 297.119,A -85,B 0,C 180,E1 -29506.969,E2 -29506.969} C_VEL
LIN {X 0,Y 126.069,Z 293.291,A -85,B 0,C 180,E1 -29510.979,E2 -29510.979} C_VEL
LIN {X 0,Y 125.495,Z 291.22,A -85,B 0,C 180,E1 -29513.972,E2 -29513.972} C_VEL
LIN {X 0,Y 125.116,Z 288.738,A -85,B 0,C 180,E1 -29520,E2 -29520} C_VEL
LIN {X 0,Y 125.65,Z 291.73,A -85,B 0,C 180,E1 -29526.826,E2 -29526.826} C_VEL
LIN {X 0,Y 126.608,Z 295.141,A -85,B 0,C 180,E1 -29531,E2 -29531} C_VEL
LIN {X 0,Y 127.234,Z 297.172,A -85,B 0,C 180,E1 -29532.967,E2 -29532.967} C_VEL
LIN {X 0,Y 124.578,Z 310.028,A -85,B 0,C 180,E1 -29533.455,E2 -29533.455} C_VEL
LIN {X 0,Y 120.498,Z 322.95,A -85,B 0,C 180,E1 -29534.165,E2 -29534.165} C_VEL
LIN {X 0,Y 115.52,Z 334.541,A -85,B 0,C 180,E1 -29535.028,E2 -29535.028} C_VEL
LIN {X 0,Y 108.948,Z 346.424,A -85,B 0,C 180,E1 -29536.35,E2 -29536.35} C_VEL
LIN {X 0,Y 101.645,Z 357.025,A -85,B 0,C 180,E1 -29538.062,E2 -29538.062} C_VEL
LIN {X 0,Y 93.651,Z 366.577,A -85,B 0,C 180,E1 -29540.27,E2 -29540.27} C_VEL
LIN {X 0,Y 84.286,Z 375.769,A -85,B 0,C 180,E1 -29543.477,E2 -29543.477} C_VEL
LIN {X 0,Y 75.045,Z 383.385,A -85,B 0,C 180,E1 -29547.747,E2 -29547.747} C_VEL
LIN {X 0,Y 66.835,Z 389.096,A -85,B 0,C 180,E1 -29552.726,E2 -29552.726} C_VEL
LIN {X 0,Y 58.919,Z 393.782,A -85,B 0,C 180,E1 -29559.162,E2 -29559.162} C_VEL
LIN {X 0,Y 51.919,Z 397.359,A -85,B 0,C 180,E1 -29567.401,E2 -29567.401} C_VEL
LIN {X 0,Y 48.065,Z 399.202,A -85,B 0,C 180,E1 -29574.202,E2 -29574.202} C_VEL
LIN {X 0,Y 42.756,Z 401.573,A -85,B 0,C 180,E1 -29590.803,E2 -29590.803} C_VEL
LIN {X 0,Y 41.481,Z 402.174,A -85,B 0,C 180,E1 -29600.241,E2 -29600.241} C_VEL
LIN {X 0,Y 41.213,Z 402.381,A -85,B 0,C 180,E1 -29609.996,E2 -29609.996} C_VEL
LIN {X 0,Y 41.48,Z 402.153,A -85,B 0,C 180,E1 -29619.75,E2 -29619.75} C_VEL
LIN {X 0,Y 42.756,Z 401.539,A -85,B 0,C 180,E1 -29629.188,E2 -29629.188} C_VEL
LIN {X 0,Y 44.98,Z 400.538,A -85,B 0,C 180,E1 -29637.947,E2 -29637.947} C_VEL
LIN {X 0,Y 48.066,Z 399.135,A -85,B 0,C 180,E1 -29645.788,E2 -29645.788} C_VEL
LIN {X 0,Y 54.133,Z 396.197,A -85,B 0,C 180,E1 -29655.56,E2 -29655.56} C_VEL
LIN {X 0,Y 61.431,Z 392.225,A -85,B 0,C 180,E1 -29663.204,E2 -29663.204} C_VEL
LIN {X 0,Y 71.029,Z 386.115,A -85,B 0,C 180,E1 -29669.964,E2 -29669.964} C_VEL
LIN {X 0,Y 79.729,Z 379.441,A -85,B 0,C 180,E1 -29674.618,E2 -29674.618} C_VEL
LIN {X 0,Y 88.923,Z 371.165,A -85,B 0,C 180,E1 -29678.218,E2 -29678.218} C_VEL
LIN {X 0,Y 96.816,Z 362.667,A -85,B 0,C 180,E1 -29680.671,E2 -29680.671} C_VEL
LIN {X 0,Y 104.86,Z 352.168,A -85,B 0,C 180,E1 -29682.751,E2 -29682.751} C_VEL
LIN {X 0,Y 112.228,Z 340.342,A -85,B 0,C 180,E1 -29684.316,E2 -29684.316} C_VEL
LIN {X 0,Y 118.307,Z 327.661,A -85,B 0,C 180,E1 -29685.477,E2 -29685.477} C_VEL
LIN {X 0,Y 122.968,Z 314.663,A -85,B 0,C 180,E1 -29686.302,E2 -29686.302} C_VEL
LIN {X 0,Y 126.156,Z 301.598,A -85,B 0,C 180,E1 -29686.818,E2 -29686.818} C_VEL
LIN {X 0,Y 126.924,Z 296.86,A -85,B 0,C 180,E1 -29687.069,E2 -29687.069} C_VEL
LIN {X 0,Y 125.804,Z 293.086,A -85,B 0,C 180,E1 -29690.96,E2 -29690.96} C_VEL
LIN {X 0,Y 125.199,Z 291.025,A -85,B 0,C 180,E1 -29693.958,E2 -29693.958} C_VEL
LIN {X 0,Y 124.83,Z 288.204,A -85,B 0,C 180,E1 -29700,E2 -29700} C_VEL
LIN {X 0,Y 125.466,Z 291.896,A -85,B 0,C 180,E1 -29707.645,E2 -29707.645} C_VEL
LIN {X 0,Y 126.353,Z 294.956,A -85,B 0,C 180,E1 -29711.328,E2 -29711.328} C_VEL
LIN {X 0,Y 126.939,Z 296.915,A -85,B 0,C 180,E1 -29713.177,E2 -29713.177} C_VEL
LIN {X 0,Y 124.183,Z 309.999,A -85,B 0,C 180,E1 -29713.682,E2 -29713.682} C_VEL
LIN {X 0,Y 120.713,Z 321.146,A -85,B 0,C 180,E1 -29714.306,E2 -29714.306} C_VEL
LIN {X 0,Y 115.656,Z 333.296,A -85,B 0,C 180,E1 -29715.286,E2 -29715.286} C_VEL
LIN {X 0,Y 115.043,Z 334.568,A -85,B 0,C 180,E1 -29715.395,E2 -29715.395} C_VEL
LIN {X 0,Y 112.213,Z 339.754,A -85,B 0,C 180,E1 -29715.576,E2 -29715.576} C_VEL
LIN {X 0,Y 106.601,Z 347.898,A -85,B 0,C 180,E1 -29715.144,E2 -29715.144} C_VEL
LIN {X 0,Y 100.387,Z 355.592,A -85,B 0,C 180,E1 -29714.806,E2 -29714.806} C_VEL
LIN {X 0,Y 96.602,Z 360.066,A -85,B 0,C 180,E1 -29715.232,E2 -29715.232} C_VEL
LIN {X 0,Y 88.341,Z 369.008,A -85,B 0,C 180,E1 -29717.33,E2 -29717.33} C_VEL
LIN {X 0,Y 78.799,Z 377.628,A -85,B 0,C 180,E1 -29720.54,E2 -29720.54} C_VEL
LIN {X 0,Y 69.546,Z 384.504,A -85,B 0,C 180,E1 -29724.572,E2 -29724.572} C_VEL
LIN {X 0,Y 60.629,Z 390.011,A -85,B 0,C 180,E1 -29729.621,E2 -29729.621} C_VEL
LIN {X 0,Y 52.282,Z 394.333,A -85,B 0,C 180,E1 -29736.247,E2 -29736.247} C_VEL
LIN {X 0,Y 47.248,Z 396.62,A -85,B 0,C 180,E1 -29741.956,E2 -29741.956} C_VEL
LIN {X 0,Y 42.826,Z 398.476,A -85,B 0,C 180,E1 -29748.979,E2 -29748.979} C_VEL
LIN {X 0,Y 39.114,Z 399.869,A -85,B 0,C 180,E1 -29757.388,E2 -29757.388} C_VEL
LIN {X 0,Y 36.32,Z 400.86,A -85,B 0,C 180,E1 -29767.238,E2 -29767.238} C_VEL
LIN {X 0,Y 34.188,Z 401.691,A -85,B 0,C 180,E1 -29790.005,E2 -29790.005} C_VEL
LIN {X 0,Y 34.603,Z 401.492,A -85,B 0,C 180,E1 -29801.723,E2 -29801.723} C_VEL
LIN {X 0,Y 36.321,Z 400.9,A -85,B 0,C 180,E1 -29812.772,E2 -29812.772} C_VEL
LIN {X 0,Y 42.819,Z 398.557,A -85,B 0,C 180,E1 -29831.04,E2 -29831.04} C_VEL
LIN {X 0,Y 49.69,Z 395.669,A -85,B 0,C 180,E1 -29841.073,E2 -29841.073} C_VEL
LIN {X 0,Y 57.741,Z 391.752,A -85,B 0,C 180,E1 -29848.435,E2 -29848.435} C_VEL
LIN {X 0,Y 66.469,Z 386.703,A -85,B 0,C 180,E1 -29853.995,E2 -29853.995} C_VEL
LIN {X 0,Y 75.622,Z 380.343,A -85,B 0,C 180,E1 -29858.339,E2 -29858.339} C_VEL
LIN {X 0,Y 85.067,Z 372.394,A -85,B 0,C 180,E1 -29861.824,E2 -29861.824} C_VEL
LIN {X 0,Y 94.846,Z 362.505,A -85,B 0,C 180,E1 -29864.429,E2 -29864.429} C_VEL
LIN {X 0,Y 103.105,Z 352.116,A -85,B 0,C 180,E1 -29866.248,E2 -29866.248} C_VEL
LIN {X 0,Y 110.608,Z 340.406,A -85,B 0,C 180,E1 -29867.668,E2 -29867.668} C_VEL
LIN {X 0,Y 116.691,Z 328.206,A -85,B 0,C 180,E1 -29868.687,E2 -29868.687} C_VEL
LIN {X 0,Y 121.535,Z 315.217,A -85,B 0,C 180,E1 -29869.438,E2 -29869.438} C_VEL
LIN {X 0,Y 124.885,Z 302.279,A -85,B 0,C 180,E1 -29869.929,E2 -29869.929} C_VEL
LIN {X 0,Y 124.974,Z 301.52,A -85,B 0,C 180,E1 -29870.083,E2 -29870.083} C_VEL
LIN {X 0,Y 124.367,Z 298.208,A -85,B 0,C 180,E1 -29874.324,E2 -29874.324} C_VEL
LIN {X 0,Y 124.146,Z 295.912,A -85,B 0,C 180,E1 -29880,E2 -29880} C_VEL
LIN {X 0,Y 124.444,Z 298.709,A -85,B 0,C 180,E1 -29886.282,E2 -29886.282} C_VEL
LIN {X 0,Y 125.011,Z 301.634,A -85,B 0,C 180,E1 -29889.914,E2 -29889.914} C_VEL
LIN {X 0,Y 121.926,Z 314.229,A -85,B 0,C 180,E1 -29890.398,E2 -29890.398} C_VEL
LIN {X 0,Y 117.29,Z 327.055,A -85,B 0,C 180,E1 -29891.095,E2 -29891.095} C_VEL
LIN {X 0,Y 111.361,Z 339.297,A -85,B 0,C 180,E1 -29891.983,E2 -29891.983} C_VEL
LIN {X 0,Y 104.665,Z 350.186,A -85,B 0,C 180,E1 -29893.184,E2 -29893.184} C_VEL
LIN {X 0,Y 96.366,Z 361.01,A -85,B 0,C 180,E1 -29894.909,E2 -29894.909} C_VEL
LIN {X 0,Y 88.164,Z 369.803,A -85,B 0,C 180,E1 -29896.945,E2 -29896.945} C_VEL
LIN {X 0,Y 78.536,Z 378.368,A -85,B 0,C 180,E1 -29900.009,E2 -29900.009} C_VEL
LIN {X 0,Y 69.255,Z 385.223,A -85,B 0,C 180,E1 -29904.029,E2 -29904.029} C_VEL
LIN {X 0,Y 60.325,Z 390.713,A -85,B 0,C 180,E1 -29909.097,E2 -29909.097} C_VEL
LIN {X 0,Y 52.007,Z 395.016,A -85,B 0,C 180,E1 -29915.821,E2 -29915.821} C_VEL
LIN {X 0,Y 46.93,Z 397.295,A -85,B 0,C 180,E1 -29921.511,E2 -29921.511} C_VEL
LIN {X 0,Y 42.479,Z 399.138,A -85,B 0,C 180,E1 -29928.56,E2 -29928.56} C_VEL
LIN {X 0,Y 36.103,Z 401.508,A -85,B 0,C 180,E1 -29947.083,E2 -29947.083} C_VEL
LIN {X 0,Y 34.506,Z 402.109,A -85,B 0,C 180,E1 -29958.243,E2 -29958.243} C_VEL
LIN {X 0,Y 34.108,Z 402.316,A -85,B 0,C 180,E1 -29969.995,E2 -29969.995} C_VEL
LIN {X 0,Y 34.505,Z 402.088,A -85,B 0,C 180,E1 -29981.747,E2 -29981.747} C_VEL
LIN {X 0,Y 36.103,Z 401.473,A -85,B 0,C 180,E1 -29992.907,E2 -29992.907} C_VEL
LIN {X 0,Y 38.819,Z 400.472,A -85,B 0,C 180,E1 -30002.891,E2 -30002.891} C_VEL
LIN {X 0,Y 42.48,Z 399.069,A -85,B 0,C 180,E1 -30011.429,E2 -30011.429} C_VEL
LIN {X 0,Y 49.416,Z 396.131,A -85,B 0,C 180,E1 -30021.457,E2 -30021.457} C_VEL
LIN {X 0,Y 57.444,Z 392.158,A -85,B 0,C 180,E1 -30028.909,E2 -30028.909} C_VEL
LIN {X 0,Y 66.246,Z 387.048,A -85,B 0,C 180,E1 -30034.381,E2 -30034.381} C_VEL
LIN {X 0,Y 75.374,Z 380.607,A -85,B 0,C 180,E1 -30038.804,E2 -30038.804} C_VEL
LIN {X 0,Y 84.914,Z 372.584,A -85,B 0,C 180,E1 -30042.13,E2 -30042.13} C_VEL
LIN {X 0,Y 93.053,Z 364.404,A -85,B 0,C 180,E1 -30044.346,E2 -30044.346} C_VEL
LIN {X 0,Y 101.303,Z 354.423,A -85,B 0,C 180,E1 -30046.218,E2 -30046.218} C_VEL
LIN {X 0,Y 108.004,Z 344.556,A -85,B 0,C 180,E1 -30047.428,E2 -30047.428} C_VEL
LIN {X 0,Y 114.723,Z 332.059,A -85,B 0,C 180,E1 -30048.556,E2 -30048.556} C_VEL
